LIN {X 0,Y 468.958,Z 580.155,A -85,B 0,C 180,E1 7791.266,E2 7791.266} C_VEL
LIN {X 0,Y 471.631,Z 601.526,A -85,B 0,C 180,E1 7791.982,E2 7791.982} C_VEL
LIN {X 0,Y 472.199,Z 602.706,A -85,B 0,C 180,E1 7792.061,E2 7792.061} C_VEL
LIN {X 0,Y 474.146,Z 606.908,A -85,B 0,C 180,E1 7792.333,E2 7792.333} C_VEL
LIN {X 0,Y 471.167,Z 650.181,A -85,B 0,C 180,E1 7793.72,E2 7793.72} C_VEL
LIN {X 0,Y 467.516,Z 690.525,A -85,B 0,C 180,E1 7795.792,E2 7795.792} C_VEL
LIN {X 0,Y 463.415,Z 728.527,A -85,B 0,C 180,E1 7798.596,E2 7798.596} C_VEL
LIN {X 0,Y 459.337,Z 761.729,A -85,B 0,C 180,E1 7801.949,E2 7801.949} C_VEL
LIN {X 0,Y 455.596,Z 791.466,A -85,B 0,C 180,E1 7805.971,E2 7805.971} C_VEL
LIN {X 0,Y 453.022,Z 813.983,A -85,B 0,C 180,E1 7810.044,E2 7810.044} C_VEL
LIN {X 0,Y 451.113,Z 833.292,A -85,B 0,C 180,E1 7814.929,E2 7814.929} C_VEL
LIN {X 0,Y 450.241,Z 846.703,A -85,B 0,C 180,E1 7819.864,E2 7819.864} C_VEL
LIN {X 0,Y 449.873,Z 853.995,A -85,B 0,C 180,E1 7824.224,E2 7824.224} C_VEL
LIN {X 0,Y 449.824,Z 857.107,A -85,B 0,C 180,E1 7828.077,E2 7828.077} C_VEL
LIN {X 0,Y 449.891,Z 857.107,A -85,B 0,C 180,E1 7831.922,E2 7831.922} C_VEL
LIN {X 0,Y 449.937,Z 852.735,A -85,B 0,C 180,E1 7836.742,E2 7836.742} C_VEL
LIN {X 0,Y 450.323,Z 843.318,A -85,B 0,C 180,E1 7841.6,E2 7841.6} C_VEL
LIN {X 0,Y 451.564,Z 828.297,A -85,B 0,C 180,E1 7846.503,E2 7846.503} C_VEL
LIN {X 0,Y 453.78,Z 807.486,A -85,B 0,C 180,E1 7851.27,E2 7851.27} C_VEL
LIN {X 0,Y 456.823,Z 782.083,A -85,B 0,C 180,E1 7855.434,E2 7855.434} C_VEL
LIN {X 0,Y 460.733,Z 750.709,A -85,B 0,C 180,E1 7859.294,E2 7859.294} C_VEL
LIN {X 0,Y 464.827,Z 716.248,A -85,B 0,C 180,E1 7862.435,E2 7862.435} C_VEL
LIN {X 0,Y 468.904,Z 677.165,A -85,B 0,C 180,E1 7865.008,E2 7865.008} C_VEL
LIN {X 0,Y 472.359,Z 635.769,A -85,B 0,C 180,E1 7866.854,E2 7866.854} C_VEL
LIN {X 0,Y 474.176,Z 604.683,A -85,B 0,C 180,E1 7867.761,E2 7867.761} C_VEL
LIN {X 0,Y 463.084,Z 582.313,A -85,B 0,C 180,E1 7869.225,E2 7869.225} C_VEL
LIN {X 0,Y 450.506,Z 554.48,A -85,B 0,C 180,E1 7870.935,E2 7870.935} C_VEL
LIN {X 0,Y 448.762,Z 549.53,A -85,B 0,C 180,E1 7871.266,E2 7871.266} C_VEL
LIN {X 0,Y 448.738,Z 549.53,A -85,B 0,C 180,E1 7877.741,E2 7877.741} C_VEL
LIN {X 0,Y 448.735,Z 549.53,A -85,B 0,C 180,E1 7883.819,E2 7883.819} C_VEL
LIN {X 0,Y 448.758,Z 549.53,A -85,B 0,C 180,E1 7889.713,E2 7889.713} C_VEL
LIN {X 0,Y 449.087,Z 549.53,A -85,B 0,C 180,E1 7895.084,E2 7895.084} C_VEL
LIN {X 0,Y 455.62,Z 577.259,A -85,B 0,C 180,E1 7895.913,E2 7895.913} C_VEL
LIN {X 0,Y 455.731,Z 612.964,A -85,B 0,C 180,E1 7896.707,E2 7896.707} C_VEL
LIN {X 0,Y 455.247,Z 640.891,A -85,B 0,C 180,E1 7898.053,E2 7898.053} C_VEL
LIN {X 0,Y 454.424,Z 665.309,A -85,B 0,C 180,E1 7899.978,E2 7899.978} C_VEL
LIN {X 0,Y 453.379,Z 686.918,A -85,B 0,C 180,E1 7902.574,E2 7902.574} C_VEL
LIN {X 0,Y 452.429,Z 703.348,A -85,B 0,C 180,E1 7905.55,E2 7905.55} C_VEL
LIN {X 0,Y 451.8,Z 714.901,A -85,B 0,C 180,E1 7908.932,E2 7908.932} C_VEL
LIN {X 0,Y 451.334,Z 720.778,A -85,B 0,C 180,E1 7912.319,E2 7912.319} C_VEL
LIN {X 0,Y 451.289,Z 721.854,A -85,B 0,C 180,E1 7914.247,E2 7914.247} C_VEL
LIN {X 0,Y 451.353,Z 719.256,A -85,B 0,C 180,E1 7918.088,E2 7918.088} C_VEL
LIN {X 0,Y 451.552,Z 711.787,A -85,B 0,C 180,E1 7921.441,E2 7921.441} C_VEL
LIN {X 0,Y 452.123,Z 698.574,A -85,B 0,C 180,E1 7924.791,E2 7924.791} C_VEL
LIN {X 0,Y 453.034,Z 679.581,A -85,B 0,C 180,E1 7927.902,E2 7927.902} C_VEL
LIN {X 0,Y 454.147,Z 656.595,A -85,B 0,C 180,E1 7930.414,E2 7930.414} C_VEL
LIN {X 0,Y 455.092,Z 630.622,A -85,B 0,C 180,E1 7932.301,E2 7932.301} C_VEL
LIN {X 0,Y 455.759,Z 601.099,A -85,B 0,C 180,E1 7933.569,E2 7933.569} C_VEL
LIN {X 0,Y 455.219,Z 572.995,A -85,B 0,C 180,E1 7934.176,E2 7934.176} C_VEL
LIN {X 0,Y 449.385,Z 549.53,A -85,B 0,C 180,E1 7934.829,E2 7934.829} C_VEL
LIN {X 0,Y 449.088,Z 549.53,A -85,B 0,C 180,E1 7941.697,E2 7941.697} C_VEL
LIN {X 0,Y 448.832,Z 549.53,A -85,B 0,C 180,E1 7948.085,E2 7948.085} C_VEL
LIN {X 0,Y 448.654,Z 549.53,A -85,B 0,C 180,E1 7954.88,E2 7954.88} C_VEL
LIN {X 0,Y 448.63,Z 549.53,A -85,B 0,C 180,E1 7959.73,E2 7959.73} C_VEL
LIN {X 0,Y 448.64,Z 549.53,A -85,B 0,C 180,E1 7965.056,E2 7965.056} C_VEL
LIN {X 0,Y 448.75,Z 549.53,A -85,B 0,C 180,E1 7970.67,E2 7970.67} C_VEL
LIN {X 0,Y 448.66,Z 549.53,A -85,B 0,C 180,E1 7977.439,E2 7977.439} C_VEL
LIN {X 0,Y 448.809,Z 550.244,A -85,B 0,C 180,E1 7978.288,E2 7978.288} C_VEL
LIN {X 0,Y 466.178,Z 592.56,A -85,B 0,C 180,E1 7981.008,E2 7981.008} C_VEL
LIN {X 0,Y 467.014,Z 599.43,A -85,B 0,C 180,E1 7981.357,E2 7981.357} C_VEL
LIN {X 0,Y 464.255,Z 634.875,A -85,B 0,C 180,E1 7983.149,E2 7983.149} C_VEL
LIN {X 0,Y 460.847,Z 669.201,A -85,B 0,C 180,E1 7985.708,E2 7985.708} C_VEL
LIN {X 0,Y 457.423,Z 699.289,A -85,B 0,C 180,E1 7988.847,E2 7988.847} C_VEL
LIN {X 0,Y 454.361,Z 725.705,A -85,B 0,C 180,E1 7992.607,E2 7992.607} C_VEL
LIN {X 0,Y 452.034,Z 746.654,A -85,B 0,C 180,E1 7996.731,E2 7996.731} C_VEL
LIN {X 0,Y 450.782,Z 761.886,A -85,B 0,C 180,E1 8000.97,E2 8000.97} C_VEL
LIN {X 0,Y 450.248,Z 771.956,A -85,B 0,C 180,E1 8005.193,E2 8005.193} C_VEL
LIN {X 0,Y 450.095,Z 778.035,A -85,B 0,C 180,E1 8010,E2 8010} C_VEL
LIN {X 0,Y 449.947,Z 778.916,A -85,B 0,C 180,E1 8013.847,E2 8013.847} C_VEL
LIN {X 0,Y 450.055,Z 775.148,A -85,B 0,C 180,E1 8018.76,E2 8018.76} C_VEL
LIN {X 0,Y 450.524,Z 765.71,A -85,B 0,C 180,E1 8023.562,E2 8023.562} C_VEL
LIN {X 0,Y 451.729,Z 751.367,A -85,B 0,C 180,E1 8028.026,E2 8028.026} C_VEL
LIN {X 0,Y 453.702,Z 731.868,A -85,B 0,C 180,E1 8032.233,E2 8032.233} C_VEL
LIN {X 0,Y 456.508,Z 707.237,A -85,B 0,C 180,E1 8036.053,E2 8036.053} C_VEL
LIN {X 0,Y 459.807,Z 678.331,A -85,B 0,C 180,E1 8039.359,E2 8039.359} C_VEL
LIN {X 0,Y 463.326,Z 644.876,A -85,B 0,C 180,E1 8042.126,E2 8042.126} C_VEL
LIN {X 0,Y 466.437,Z 608.507,A -85,B 0,C 180,E1 8044.2,E2 8044.2} C_VEL
LIN {X 0,Y 466.662,Z 594.193,A -85,B 0,C 180,E1 8044.838,E2 8044.838} C_VEL
LIN {X 0,Y 453.477,Z 560.1,A -85,B 0,C 180,E1 8047.08,E2 8047.08} C_VEL
LIN {X 0,Y 448.888,Z 549.53,A -85,B 0,C 180,E1 8047.902,E2 8047.902} C_VEL
LIN {X 0,Y 448.628,Z 549.53,A -85,B 0,C 180,E1 8055.054,E2 8055.054} C_VEL
LIN {X 0,Y 448.8,Z 549.53,A -85,B 0,C 180,E1 8060.663,E2 8060.663} C_VEL
LIN {X 0,Y 448.849,Z 549.53,A -85,B 0,C 180,E1 8067.202,E2 8067.202} C_VEL
LIN {X 0,Y 448.843,Z 549.53,A -85,B 0,C 180,E1 8074.078,E2 8074.078} C_VEL
LIN {X 0,Y 449.012,Z 549.53,A -85,B 0,C 180,E1 8078.739,E2 8078.739} C_VEL
LIN {X 0,Y 454.538,Z 576.815,A -85,B 0,C 180,E1 8079.412,E2 8079.412} C_VEL
LIN {X 0,Y 454.441,Z 624.708,A -85,B 0,C 180,E1 8080.368,E2 8080.368} C_VEL
LIN {X 0,Y 453.943,Z 650.535,A -85,B 0,C 180,E1 8081.607,E2 8081.607} C_VEL
LIN {X 0,Y 453.192,Z 674.327,A -85,B 0,C 180,E1 8083.554,E2 8083.554} C_VEL
LIN {X 0,Y 452.281,Z 694.707,A -85,B 0,C 180,E1 8086.171,E2 8086.171} C_VEL
LIN {X 0,Y 451.81,Z 708.538,A -85,B 0,C 180,E1 8088.923,E2 8088.923} C_VEL
LIN {X 0,Y 451.452,Z 717.552,A -85,B 0,C 180,E1 8091.839,E2 8091.839} C_VEL
LIN {X 0,Y 451.351,Z 721.412,A -85,B 0,C 180,E1 8094.239,E2 8094.239} C_VEL
LIN {X 0,Y 451.349,Z 722.421,A -85,B 0,C 180,E1 8096.162,E2 8096.162} C_VEL
LIN {X 0,Y 451.475,Z 720.452,A -85,B 0,C 180,E1 8099.038,E2 8099.038} C_VEL
LIN {X 0,Y 451.94,Z 712.572,A -85,B 0,C 180,E1 8102.388,E2 8102.388} C_VEL
LIN {X 0,Y 452.653,Z 700.047,A -85,B 0,C 180,E1 8105.256,E2 8105.256} C_VEL
LIN {X 0,Y 453.465,Z 681.764,A -85,B 0,C 180,E1 8107.886,E2 8107.886} C_VEL
LIN {X 0,Y 454.249,Z 659.647,A -85,B 0,C 180,E1 8109.914,E2 8109.914} C_VEL
LIN {X 0,Y 454.624,Z 634.95,A -85,B 0,C 180,E1 8111.285,E2 8111.285} C_VEL
LIN {X 0,Y 454.621,Z 605.314,A -85,B 0,C 180,E1 8112.05,E2 8112.05} C_VEL
LIN {X 0,Y 454.181,Z 569.256,A -85,B 0,C 180,E1 8112.708,E2 8112.708} C_VEL
LIN {X 0,Y 449.327,Z 549.53,A -85,B 0,C 180,E1 8113.328,E2 8113.328} C_VEL
LIN {X 0,Y 449.048,Z 549.53,A -85,B 0,C 180,E1 8119.773,E2 8119.773} C_VEL
LIN {X 0,Y 448.861,Z 549.53,A -85,B 0,C 180,E1 8125.911,E2 8125.911} C_VEL
LIN {X 0,Y 448.646,Z 549.53,A -85,B 0,C 180,E1 8132.757,E2 8132.757} C_VEL
LIN {X 0,Y 448.756,Z 549.53,A -85,B 0,C 180,E1 8139.331,E2 8139.331} C_VEL
LIN {X 0,Y 448.66,Z 549.53,A -85,B 0,C 180,E1 8145.058,E2 8145.058} C_VEL
LIN {X 0,Y 448.725,Z 549.68,A -85,B 0,C 180,E1 8148.7,E2 8148.7} C_VEL
LIN {X 0,Y 453.525,Z 559.924,A -85,B 0,C 180,E1 8149.401,E2 8149.401} C_VEL
LIN {X 0,Y 470.3,Z 599.601,A -85,B 0,C 180,E1 8151.819,E2 8151.819} C_VEL
LIN {X 0,Y 472.199,Z 602.706,A -85,B 0,C 180,E1 8152.061,E2 8152.061} C_VEL
LIN {X 0,Y 472.315,Z 609.467,A -85,B 0,C 180,E1 8152.253,E2 8152.253} C_VEL
LIN {X 0,Y 466.587,Z 624.047,A -85,B 0,C 180,E1 8152.272,E2 8152.272} C_VEL
LIN {X 0,Y 466.404,Z 625.593,A -85,B 0,C 180,E1 8152.315,E2 8152.315} C_VEL
LIN {X 0,Y 462.996,Z 666.329,A -85,B 0,C 180,E1 8153.961,E2 8153.961} C_VEL
LIN {X 0,Y 458.94,Z 704.99,A -85,B 0,C 180,E1 8156.282,E2 8156.282} C_VEL
LIN {X 0,Y 454.394,Z 742.555,A -85,B 0,C 180,E1 8159.469,E2 8159.469} C_VEL
LIN {X 0,Y 450.434,Z 773.095,A -85,B 0,C 180,E1 8162.997,E2 8162.997} C_VEL
LIN {X 0,Y 446.719,Z 801.611,A -85,B 0,C 180,E1 8167.4,E2 8167.4} C_VEL
LIN {X 0,Y 444.117,Z 824.449,A -85,B 0,C 180,E1 8172.191,E2 8172.191} C_VEL
LIN {X 0,Y 442.649,Z 840.782,A -85,B 0,C 180,E1 8177.196,E2 8177.196} C_VEL
LIN {X 0,Y 442.08,Z 851.261,A -85,B 0,C 180,E1 8182.151,E2 8182.151} C_VEL
LIN {X 0,Y 441.884,Z 855.94,A -85,B 0,C 180,E1 8186.083,E2 8186.083} C_VEL
LIN {X 0,Y 441.939,Z 857.5,A -85,B 0,C 180,E1 8190,E2 8190} C_VEL
LIN {X 0,Y 441.903,Z 855.94,A -85,B 0,C 180,E1 8193.916,E2 8193.916} C_VEL
LIN {X 0,Y 442.182,Z 849.486,A -85,B 0,C 180,E1 8198.894,E2 8198.894} C_VEL
LIN {X 0,Y 442.989,Z 836.944,A -85,B 0,C 180,E1 8204.165,E2 8204.165} C_VEL
LIN {X 0,Y 444.463,Z 821.337,A -85,B 0,C 180,E1 8208.564,E2 8208.564} C_VEL
LIN {X 0,Y 447.229,Z 797.324,A -85,B 0,C 180,E1 8213.359,E2 8213.359} C_VEL
LIN {X 0,Y 451.125,Z 768.092,A -85,B 0,C 180,E1 8217.665,E2 8217.665} C_VEL
LIN {X 0,Y 455.3,Z 736.094,A -85,B 0,C 180,E1 8221.167,E2 8221.167} C_VEL
LIN {X 0,Y 459.557,Z 700.748,A -85,B 0,C 180,E1 8224.023,E2 8224.023} C_VEL
LIN {X 0,Y 463.565,Z 661.836,A -85,B 0,C 180,E1 8226.279,E2 8226.279} C_VEL
LIN {X 0,Y 466.918,Z 621.282,A -85,B 0,C 180,E1 8227.832,E2 8227.832} C_VEL
LIN {X 0,Y 467.172,Z 607.41,A -85,B 0,C 180,E1 8228.257,E2 8228.257} C_VEL
LIN {X 0,Y 455.657,Z 582.229,A -85,B 0,C 180,E1 8229.897,E2 8229.897} C_VEL
LIN {X 0,Y 442.976,Z 554.912,A -85,B 0,C 180,E1 8231.669,E2 8231.669} C_VEL
LIN {X 0,Y 440.83,Z 549.53,A -85,B 0,C 180,E1 8232.063,E2 8232.063} C_VEL
LIN {X 0,Y 440.77,Z 549.53,A -85,B 0,C 180,E1 8238.874,E2 8238.874} C_VEL
LIN {X 0,Y 440.809,Z 549.53,A -85,B 0,C 180,E1 8245.253,E2 8245.253} C_VEL
LIN {X 0,Y 440.892,Z 549.53,A -85,B 0,C 180,E1 8251.374,E2 8251.374} C_VEL
LIN {X 0,Y 441.126,Z 549.809,A -85,B 0,C 180,E1 8254.732,E2 8254.732} C_VEL
LIN {X 0,Y 448.163,Z 578.479,A -85,B 0,C 180,E1 8255.616,E2 8255.616} C_VEL
LIN {X 0,Y 448.252,Z 614.662,A -85,B 0,C 180,E1 8256.441,E2 8256.441} C_VEL
LIN {X 0,Y 447.746,Z 642.172,A -85,B 0,C 180,E1 8257.782,E2 8257.782} C_VEL
LIN {X 0,Y 446.889,Z 666.849,A -85,B 0,C 180,E1 8259.755,E2 8259.755} C_VEL
LIN {X 0,Y 445.835,Z 687.649,A -85,B 0,C 180,E1 8262.269,E2 8262.269} C_VEL
LIN {X 0,Y 444.822,Z 704.385,A -85,B 0,C 180,E1 8265.297,E2 8265.297} C_VEL
LIN {X 0,Y 444.113,Z 716.107,A -85,B 0,C 180,E1 8268.738,E2 8268.738} C_VEL
LIN {X 0,Y 443.58,Z 722.102,A -85,B 0,C 180,E1 8272.184,E2 8272.184} C_VEL
LIN {X 0,Y 443.521,Z 723.232,A -85,B 0,C 180,E1 8274.146,E2 8274.146} C_VEL
LIN {X 0,Y 443.592,Z 720.65,A -85,B 0,C 180,E1 8278.055,E2 8278.055} C_VEL
LIN {X 0,Y 443.789,Z 713.177,A -85,B 0,C 180,E1 8281.466,E2 8281.466} C_VEL
LIN {X 0,Y 444.372,Z 699.941,A -85,B 0,C 180,E1 8284.875,E2 8284.875} C_VEL
LIN {X 0,Y 445.316,Z 680.911,A -85,B 0,C 180,E1 8288.04,E2 8288.04} C_VEL
LIN {X 0,Y 446.47,Z 657.872,A -85,B 0,C 180,E1 8290.595,E2 8290.595} C_VEL
LIN {X 0,Y 447.489,Z 630.925,A -85,B 0,C 180,E1 8292.567,E2 8292.567} C_VEL
LIN {X 0,Y 448.18,Z 601.127,A -85,B 0,C 180,E1 8293.844,E2 8293.844} C_VEL
LIN {X 0,Y 447.583,Z 573.933,A -85,B 0,C 180,E1 8294.438,E2 8294.438} C_VEL
LIN {X 0,Y 441.441,Z 549.53,A -85,B 0,C 180,E1 8295.121,E2 8295.121} C_VEL
LIN {X 0,Y 441.119,Z 549.53,A -85,B 0,C 180,E1 8302.11,E2 8302.11} C_VEL
LIN {X 0,Y 440.911,Z 549.53,A -85,B 0,C 180,E1 8308.635,E2 8308.635} C_VEL
LIN {X 0,Y 440.731,Z 549.53,A -85,B 0,C 180,E1 8315.602,E2 8315.602} C_VEL
LIN {X 0,Y 440.614,Z 549.53,A -85,B 0,C 180,E1 8321.103,E2 8321.103} C_VEL
LIN {X 0,Y 440.674,Z 549.53,A -85,B 0,C 180,E1 8326.769,E2 8326.769} C_VEL
LIN {X 0,Y 440.771,Z 549.53,A -85,B 0,C 180,E1 8331.953,E2 8331.953} C_VEL
LIN {X 0,Y 440.806,Z 550.142,A -85,B 0,C 180,E1 8337.555,E2 8337.555} C_VEL
LIN {X 0,Y 457.96,Z 591.22,A -85,B 0,C 180,E1 8340.312,E2 8340.312} C_VEL
LIN {X 0,Y 460.191,Z 600.559,A -85,B 0,C 180,E1 8340.887,E2 8340.887} C_VEL
LIN {X 0,Y 457.232,Z 636.395,A -85,B 0,C 180,E1 8342.744,E2 8342.744} C_VEL
LIN {X 0,Y 453.677,Z 669.986,A -85,B 0,C 180,E1 8345.298,E2 8345.298} C_VEL
LIN {X 0,Y 450.19,Z 698.924,A -85,B 0,C 180,E1 8348.362,E2 8348.362} C_VEL
LIN {X 0,Y 446.944,Z 725.067,A -85,B 0,C 180,E1 8352.087,E2 8352.087} C_VEL
LIN {X 0,Y 444.456,Z 746.31,A -85,B 0,C 180,E1 8356.25,E2 8356.25} C_VEL
LIN {X 0,Y 442.984,Z 762.695,A -85,B 0,C 180,E1 8360.832,E2 8360.832} C_VEL
LIN {X 0,Y 442.398,Z 772.708,A -85,B 0,C 180,E1 8365.108,E2 8365.108} C_VEL
LIN {X 0,Y 442.246,Z 778.766,A -85,B 0,C 180,E1 8370,E2 8370} C_VEL
LIN {X 0,Y 442.09,Z 779.613,A -85,B 0,C 180,E1 8373.915,E2 8373.915} C_VEL
LIN {X 0,Y 442.22,Z 775.839,A -85,B 0,C 180,E1 8378.855,E2 8378.855} C_VEL
LIN {X 0,Y 442.67,Z 767.491,A -85,B 0,C 180,E1 8383.301,E2 8383.301} C_VEL
LIN {X 0,Y 443.856,Z 753.673,A -85,B 0,C 180,E1 8387.82,E2 8387.82} C_VEL
LIN {X 0,Y 445.91,Z 734.596,A -85,B 0,C 180,E1 8392.119,E2 8392.119} C_VEL
LIN {X 0,Y 448.796,Z 710.116,A -85,B 0,C 180,E1 8396.102,E2 8396.102} C_VEL
LIN {X 0,Y 452.409,Z 680.764,A -85,B 0,C 180,E1 8399.601,E2 8399.601} C_VEL
LIN {X 0,Y 456.178,Z 647.674,A -85,B 0,C 180,E1 8402.448,E2 8402.448} C_VEL
LIN {X 0,Y 459.521,Z 612.087,A -85,B 0,C 180,E1 8404.563,E2 8404.563} C_VEL
LIN {X 0,Y 459.83,Z 596.401,A -85,B 0,C 180,E1 8405.302,E2 8405.302} C_VEL
LIN {X 0,Y 447.484,Z 564.002,A -85,B 0,C 180,E1 8407.525,E2 8407.525} C_VEL
LIN {X 0,Y 440.941,Z 549.53,A -85,B 0,C 180,E1 8408.628,E2 8408.628} C_VEL
LIN {X 0,Y 440.65,Z 549.53,A -85,B 0,C 180,E1 8415.991,E2 8415.991} C_VEL
LIN {X 0,Y 440.881,Z 549.53,A -85,B 0,C 180,E1 8421.963,E2 8421.963} C_VEL
LIN {X 0,Y 440.923,Z 549.53,A -85,B 0,C 180,E1 8426.793,E2 8426.793} C_VEL
LIN {X 0,Y 440.882,Z 549.53,A -85,B 0,C 180,E1 8433.574,E2 8433.574} C_VEL
LIN {X 0,Y 441.08,Z 549.53,A -85,B 0,C 180,E1 8438.424,E2 8438.424} C_VEL
LIN {X 0,Y 446.961,Z 578.421,A -85,B 0,C 180,E1 8439.19,E2 8439.19} C_VEL
LIN {X 0,Y 446.777,Z 625.969,A -85,B 0,C 180,E1 8440.16,E2 8440.16} C_VEL
LIN {X 0,Y 446.244,Z 652.884,A -85,B 0,C 180,E1 8441.495,E2 8441.495} C_VEL
LIN {X 0,Y 445.445,Z 676.631,A -85,B 0,C 180,E1 8443.513,E2 8443.513} C_VEL
LIN {X 0,Y 444.553,Z 695.54,A -85,B 0,C 180,E1 8445.986,E2 8445.986} C_VEL
LIN {X 0,Y 444.065,Z 709.321,A -85,B 0,C 180,E1 8448.728,E2 8448.728} C_VEL
LIN {X 0,Y 443.704,Z 717.704,A -85,B 0,C 180,E1 8451.325,E2 8451.325} C_VEL
LIN {X 0,Y 443.582,Z 722.615,A -85,B 0,C 180,E1 8454.138,E2 8454.138} C_VEL
LIN {X 0,Y 443.582,Z 723.739,A -85,B 0,C 180,E1 8456.094,E2 8456.094} C_VEL
LIN {X 0,Y 443.706,Z 721.914,A -85,B 0,C 180,E1 8459.021,E2 8459.021} C_VEL
LIN {X 0,Y 444.218,Z 714.183,A -85,B 0,C 180,E1 8462.429,E2 8462.429} C_VEL
LIN {X 0,Y 444.974,Z 701.791,A -85,B 0,C 180,E1 8465.347,E2 8465.347} C_VEL
LIN {X 0,Y 445.847,Z 683.655,A -85,B 0,C 180,E1 8468.021,E2 8468.021} C_VEL
LIN {X 0,Y 446.623,Z 661.695,A -85,B 0,C 180,E1 8470.09,E2 8470.09} C_VEL
LIN {X 0,Y 447.066,Z 635.885,A -85,B 0,C 180,E1 8471.549,E2 8471.549} C_VEL
LIN {X 0,Y 447.075,Z 605.219,A -85,B 0,C 180,E1 8472.339,E2 8472.339} C_VEL
LIN {X 0,Y 446.826,Z 571.258,A -85,B 0,C 180,E1 8472.971,E2 8472.971} C_VEL
LIN {X 0,Y 441.397,Z 549.53,A -85,B 0,C 180,E1 8473.636,E2 8473.636} C_VEL
LIN {X 0,Y 441.132,Z 549.53,A -85,B 0,C 180,E1 8479.999,E2 8479.999} C_VEL
LIN {X 0,Y 440.879,Z 549.53,A -85,B 0,C 180,E1 8486.416,E2 8486.416} C_VEL
LIN {X 0,Y 440.704,Z 549.53,A -85,B 0,C 180,E1 8493.215,E2 8493.215} C_VEL
LIN {X 0,Y 440.787,Z 549.53,A -85,B 0,C 180,E1 8498.049,E2 8498.049} C_VEL
LIN {X 0,Y 440.686,Z 549.53,A -85,B 0,C 180,E1 8504.014,E2 8504.014} C_VEL
LIN {X 0,Y 440.783,Z 549.53,A -85,B 0,C 180,E1 8507.826,E2 8507.826} C_VEL
LIN {X 0,Y 445.066,Z 559.069,A -85,B 0,C 180,E1 8508.506,E2 8508.506} C_VEL
LIN {X 0,Y 453.835,Z 578.128,A -85,B 0,C 180,E1 8509.804,E2 8509.804} C_VEL
LIN {X 0,Y 464.775,Z 604.46,A -85,B 0,C 180,E1 8511.477,E2 8511.477} C_VEL
LIN {X 0,Y 467.444,Z 608.833,A -85,B 0,C 180,E1 8511.828,E2 8511.828} C_VEL
LIN {X 0,Y 466.404,Z 625.593,A -85,B 0,C 180,E1 8512.315,E2 8512.315} C_VEL
LIN {X 0,Y 461.732,Z 642.303,A -85,B 0,C 180,E1 8512.633,E2 8512.633} C_VEL
LIN {X 0,Y 457.12,Z 656.694,A -85,B 0,C 180,E1 8512.98,E2 8512.98} C_VEL
LIN {X 0,Y 456.86,Z 658.754,A -85,B 0,C 180,E1 8513.069,E2 8513.069} C_VEL
LIN {X 0,Y 452.474,Z 700.061,A -85,B 0,C 180,E1 8515.457,E2 8515.457} C_VEL
LIN {X 0,Y 447.896,Z 737.285,A -85,B 0,C 180,E1 8518.515,E2 8518.515} C_VEL
LIN {X 0,Y 443.641,Z 768.24,A -85,B 0,C 180,E1 8521.981,E2 8521.981} C_VEL
LIN {X 0,Y 439.677,Z 796.512,A -85,B 0,C 180,E1 8526.214,E2 8526.214} C_VEL
LIN {X 0,Y 436.742,Z 820.602,A -85,B 0,C 180,E1 8531.097,E2 8531.097} C_VEL
LIN {X 0,Y 434.988,Z 838.73,A -85,B 0,C 180,E1 8536.234,E2 8536.234} C_VEL
LIN {X 0,Y 434.288,Z 849.592,A -85,B 0,C 180,E1 8541.003,E2 8541.003} C_VEL
LIN {X 0,Y 434.002,Z 855.939,A -85,B 0,C 180,E1 8546.012,E2 8546.012} C_VEL
LIN {X 0,Y 434.039,Z 857.5,A -85,B 0,C 180,E1 8550,E2 8550} C_VEL
LIN {X 0,Y 434.021,Z 855.939,A -85,B 0,C 180,E1 8553.987,E2 8553.987} C_VEL
LIN {X 0,Y 434.288,Z 849.594,A -85,B 0,C 180,E1 8558.996,E2 8558.996} C_VEL
LIN {X 0,Y 435.088,Z 837.877,A -85,B 0,C 180,E1 8564.052,E2 8564.052} C_VEL
LIN {X 0,Y 436.836,Z 819.531,A -85,B 0,C 180,E1 8569.16,E2 8569.16} C_VEL
LIN {X 0,Y 439.656,Z 796.582,A -85,B 0,C 180,E1 8573.786,E2 8573.786} C_VEL
LIN {X 0,Y 443.666,Z 768.377,A -85,B 0,C 180,E1 8578.016,E2 8578.016} C_VEL
LIN {X 0,Y 447.921,Z 737.455,A -85,B 0,C 180,E1 8581.482,E2 8581.482} C_VEL
LIN {X 0,Y 452.467,Z 702.018,A -85,B 0,C 180,E1 8584.426,E2 8584.426} C_VEL
LIN {X 0,Y 456.624,Z 663.574,A -85,B 0,C 180,E1 8586.713,E2 8586.713} C_VEL
LIN {X 0,Y 460.316,Z 621.55,A -85,B 0,C 180,E1 8588.364,E2 8588.364} C_VEL
LIN {X 0,Y 460.446,Z 610.446,A -85,B 0,C 180,E1 8588.732,E2 8588.732} C_VEL
LIN {X 0,Y 448.851,Z 583.513,A -85,B 0,C 180,E1 8590.505,E2 8590.505} C_VEL
LIN {X 0,Y 436.391,Z 557.835,A -85,B 0,C 180,E1 8592.283,E2 8592.283} C_VEL
LIN {X 0,Y 432.841,Z 549.53,A -85,B 0,C 180,E1 8592.941,E2 8592.941} C_VEL
LIN {X 0,Y 432.825,Z 549.53,A -85,B 0,C 180,E1 8598.521,E2 8598.521} C_VEL
LIN {X 0,Y 432.835,Z 549.53,A -85,B 0,C 180,E1 8603.658,E2 8603.658} C_VEL
LIN {X 0,Y 432.881,Z 549.53,A -85,B 0,C 180,E1 8610.643,E2 8610.643} C_VEL
LIN {X 0,Y 433.162,Z 549.53,A -85,B 0,C 180,E1 8614.303,E2 8614.303} C_VEL
LIN {X 0,Y 440.728,Z 579.778,A -85,B 0,C 180,E1 8615.301,E2 8615.301} C_VEL
LIN {X 0,Y 440.78,Z 616.347,A -85,B 0,C 180,E1 8616.154,E2 8616.154} C_VEL
LIN {X 0,Y 440.254,Z 645.272,A -85,B 0,C 180,E1 8617.616,E2 8617.616} C_VEL
LIN {X 0,Y 439.278,Z 670.948,A -85,B 0,C 180,E1 8619.782,E2 8619.782} C_VEL
LIN {X 0,Y 438.108,Z 691.789,A -85,B 0,C 180,E1 8622.464,E2 8622.464} C_VEL
LIN {X 0,Y 437.01,Z 708.322,A -85,B 0,C 180,E1 8625.729,E2 8625.729} C_VEL
LIN {X 0,Y 436.35,Z 718.588,A -85,B 0,C 180,E1 8629.04,E2 8629.04} C_VEL
LIN {X 0,Y 435.828,Z 723.442,A -85,B 0,C 180,E1 8632.044,E2 8632.044} C_VEL
LIN {X 0,Y 435.743,Z 724.604,A -85,B 0,C 180,E1 8634.041,E2 8634.041} C_VEL
LIN {X 0,Y 435.779,Z 723.27,A -85,B 0,C 180,E1 8637.027,E2 8637.027} C_VEL
LIN {X 0,Y 435.907,Z 717.221,A -85,B 0,C 180,E1 8640.5,E2 8640.5} C_VEL
LIN {X 0,Y 436.422,Z 705.775,A -85,B 0,C 180,E1 8643.97,E2 8643.97} C_VEL
LIN {X 0,Y 437.261,Z 688.914,A -85,B 0,C 180,E1 8647.191,E2 8647.191} C_VEL
LIN {X 0,Y 438.388,Z 667.876,A -85,B 0,C 180,E1 8649.915,E2 8649.915} C_VEL
LIN {X 0,Y 439.504,Z 642.176,A -85,B 0,C 180,E1 8652.145,E2 8652.145} C_VEL
LIN {X 0,Y 440.406,Z 613.587,A -85,B 0,C 180,E1 8653.693,E2 8653.693} C_VEL
LIN {X 0,Y 440.767,Z 580.332,A -85,B 0,C 180,E1 8654.57,E2 8654.57} C_VEL
LIN {X 0,Y 433.502,Z 549.53,A -85,B 0,C 180,E1 8655.471,E2 8655.471} C_VEL
LIN {X 0,Y 433.183,Z 549.53,A -85,B 0,C 180,E1 8662.537,E2 8662.537} C_VEL
LIN {X 0,Y 432.894,Z 549.53,A -85,B 0,C 180,E1 8669.36,E2 8669.36} C_VEL
LIN {X 0,Y 432.823,Z 549.53,A -85,B 0,C 180,E1 8673.912,E2 8673.912} C_VEL
LIN {X 0,Y 432.657,Z 549.53,A -85,B 0,C 180,E1 8679.88,E2 8679.88} C_VEL
LIN {X 0,Y 432.741,Z 549.53,A -85,B 0,C 180,E1 8685.774,E2 8685.774} C_VEL
LIN {X 0,Y 432.763,Z 549.53,A -85,B 0,C 180,E1 8691.119,E2 8691.119} C_VEL
LIN {X 0,Y 432.875,Z 550.253,A -85,B 0,C 180,E1 8696.797,E2 8696.797} C_VEL
LIN {X 0,Y 450.238,Z 590.991,A -85,B 0,C 180,E1 8699.671,E2 8699.671} C_VEL
LIN {X 0,Y 453.385,Z 601.945,A -85,B 0,C 180,E1 8700.412,E2 8700.412} C_VEL
LIN {X 0,Y 450.283,Z 637.555,A -85,B 0,C 180,E1 8702.298,E2 8702.298} C_VEL
LIN {X 0,Y 446.554,Z 670.859,A -85,B 0,C 180,E1 8704.877,E2 8704.877} C_VEL
LIN {X 0,Y 442.59,Z 701.666,A -85,B 0,C 180,E1 8708.234,E2 8708.234} C_VEL
LIN {X 0,Y 439.254,Z 727.045,A -85,B 0,C 180,E1 8711.988,E2 8711.988} C_VEL
LIN {X 0,Y 436.674,Z 748.042,A -85,B 0,C 180,E1 8716.255,E2 8716.255} C_VEL
LIN {X 0,Y 435.142,Z 764.326,A -85,B 0,C 180,E1 8720.976,E2 8720.976} C_VEL
LIN {X 0,Y 434.562,Z 773.455,A -85,B 0,C 180,E1 8725.02,E2 8725.02} C_VEL
LIN {X 0,Y 434.382,Z 779.497,A -85,B 0,C 180,E1 8730,E2 8730} C_VEL
LIN {X 0,Y 434.213,Z 780.312,A -85,B 0,C 180,E1 8733.986,E2 8733.986} C_VEL
LIN {X 0,Y 434.36,Z 776.472,A -85,B 0,C 180,E1 8738.996,E2 8738.996} C_VEL
LIN {X 0,Y 434.91,Z 767.593,A -85,B 0,C 180,E1 8743.686,E2 8743.686} C_VEL
LIN {X 0,Y 436.165,Z 753.978,A -85,B 0,C 180,E1 8748.145,E2 8748.145} C_VEL
LIN {X 0,Y 438.349,Z 734.743,A -85,B 0,C 180,E1 8752.521,E2 8752.521} C_VEL
LIN {X 0,Y 441.656,Z 709.389,A -85,B 0,C 180,E1 8756.674,E2 8756.674} C_VEL
LIN {X 0,Y 445.474,Z 680.527,A -85,B 0,C 180,E1 8760.143,E2 8760.143} C_VEL
LIN {X 0,Y 449.419,Z 647.615,A -85,B 0,C 180,E1 8762.991,E2 8762.991} C_VEL
LIN {X 0,Y 452.837,Z 612.932,A -85,B 0,C 180,E1 8765.08,E2 8765.08} C_VEL
LIN {X 0,Y 453.234,Z 599.105,A -85,B 0,C 180,E1 8765.745,E2 8765.745} C_VEL
LIN {X 0,Y 441.659,Z 568.235,A -85,B 0,C 180,E1 8767.958,E2 8767.958} C_VEL
LIN {X 0,Y 432.941,Z 549.53,A -85,B 0,C 180,E1 8769.484,E2 8769.484} C_VEL
LIN {X 0,Y 432.728,Z 549.53,A -85,B 0,C 180,E1 8775.771,E2 8775.771} C_VEL
LIN {X 0,Y 432.869,Z 549.53,A -85,B 0,C 180,E1 8781.128,E2 8781.128} C_VEL
LIN {X 0,Y 433.045,Z 549.53,A -85,B 0,C 180,E1 8786.764,E2 8786.764} C_VEL
LIN {X 0,Y 432.976,Z 549.53,A -85,B 0,C 180,E1 8793.053,E2 8793.053} C_VEL
LIN {X 0,Y 433.145,Z 549.53,A -85,B 0,C 180,E1 8798.145,E2 8798.145} C_VEL
LIN {X 0,Y 439.232,Z 577.752,A -85,B 0,C 180,E1 8798.913,E2 8798.913} C_VEL
LIN {X 0,Y 439.136,Z 627.616,A -85,B 0,C 180,E1 8799.959,E2 8799.959} C_VEL
LIN {X 0,Y 438.556,Z 654.011,A -85,B 0,C 180,E1 8801.295,E2 8801.295} C_VEL
LIN {X 0,Y 437.737,Z 677.768,A -85,B 0,C 180,E1 8803.343,E2 8803.343} C_VEL
LIN {X 0,Y 436.783,Z 697.587,A -85,B 0,C 180,E1 8806,E2 8806} C_VEL
LIN {X 0,Y 436.24,Z 712.054,A -85,B 0,C 180,E1 8809.028,E2 8809.028} C_VEL
LIN {X 0,Y 435.8,Z 721.391,A -85,B 0,C 180,E1 8812.422,E2 8812.422} C_VEL
LIN {X 0,Y 435.811,Z 725.06,A -85,B 0,C 180,E1 8816.024,E2 8816.024} C_VEL
LIN {X 0,Y 435.959,Z 723.389,A -85,B 0,C 180,E1 8819.004,E2 8819.004} C_VEL
LIN {X 0,Y 436.504,Z 715.825,A -85,B 0,C 180,E1 8822.472,E2 8822.472} C_VEL
LIN {X 0,Y 437.281,Z 703.545,A -85,B 0,C 180,E1 8825.441,E2 8825.441} C_VEL
LIN {X 0,Y 438.22,Z 685.578,A -85,B 0,C 180,E1 8828.162,E2 8828.162} C_VEL
LIN {X 0,Y 439.061,Z 663.153,A -85,B 0,C 180,E1 8830.325,E2 8830.325} C_VEL
LIN {X 0,Y 439.537,Z 637.121,A -85,B 0,C 180,E1 8831.817,E2 8831.817} C_VEL
LIN {X 0,Y 439.523,Z 604.015,A -85,B 0,C 180,E1 8832.661,E2 8832.661} C_VEL
LIN {X 0,Y 439.068,Z 571.373,A -85,B 0,C 180,E1 8833.306,E2 8833.306} C_VEL
LIN {X 0,Y 433.411,Z 549.53,A -85,B 0,C 180,E1 8834.102,E2 8834.102} C_VEL
LIN {X 0,Y 433.18,Z 549.53,A -85,B 0,C 180,E1 8840.382,E2 8840.382} C_VEL
LIN {X 0,Y 432.955,Z 549.53,A -85,B 0,C 180,E1 8846.938,E2 8846.938} C_VEL
LIN {X 0,Y 432.807,Z 549.53,A -85,B 0,C 180,E1 8853.902,E2 8853.902} C_VEL
LIN {X 0,Y 432.766,Z 549.53,A -85,B 0,C 180,E1 8859.896,E2 8859.896} C_VEL
LIN {X 0,Y 432.778,Z 549.53,A -85,B 0,C 180,E1 8866.379,E2 8866.379} C_VEL
LIN {X 0,Y 432.791,Z 549.531,A -85,B 0,C 180,E1 8866.936,E2 8866.936} C_VEL
LIN {X 0,Y 435.183,Z 555.159,A -85,B 0,C 180,E1 8867.334,E2 8867.334} C_VEL
LIN {X 0,Y 446.252,Z 577.13,A -85,B 0,C 180,E1 8869.016,E2 8869.016} C_VEL
LIN {X 0,Y 458.627,Z 608.29,A -85,B 0,C 180,E1 8871.049,E2 8871.049} C_VEL
LIN {X 0,Y 460.755,Z 612.999,A -85,B 0,C 180,E1 8871.392,E2 8871.392} C_VEL
LIN {X 0,Y 456.984,Z 657.402,A -85,B 0,C 180,E1 8873.007,E2 8873.007} C_VEL
LIN {X 0,Y 456.86,Z 658.754,A -85,B 0,C 180,E1 8873.069,E2 8873.069} C_VEL
LIN {X 0,Y 451.965,Z 674.993,A -85,B 0,C 180,E1 8873.641,E2 8873.641} C_VEL
LIN {X 0,Y 446.703,Z 690.803,A -85,B 0,C 180,E1 8874.34,E2 8874.34} C_VEL
LIN {X 0,Y 442.073,Z 727.964,A -85,B 0,C 180,E1 8877.183,E2 8877.183} C_VEL
LIN {X 0,Y 437.392,Z 760.685,A -85,B 0,C 180,E1 8880.609,E2 8880.609} C_VEL
LIN {X 0,Y 433.142,Z 789.231,A -85,B 0,C 180,E1 8884.659,E2 8884.659} C_VEL
LIN {X 0,Y 429.68,Z 814.276,A -85,B 0,C 180,E1 8889.437,E2 8889.437} C_VEL
LIN {X 0,Y 427.527,Z 834.039,A -85,B 0,C 180,E1 8894.647,E2 8894.647} C_VEL
LIN {X 0,Y 426.596,Z 847.379,A -85,B 0,C 180,E1 8899.811,E2 8899.811} C_VEL
LIN {X 0,Y 426.191,Z 853.972,A -85,B 0,C 180,E1 8903.901,E2 8903.901} C_VEL
LIN {X 0,Y 426.108,Z 857.104,A -85,B 0,C 180,E1 8907.97,E2 8907.97} C_VEL
LIN {X 0,Y 426.17,Z 857.104,A -85,B 0,C 180,E1 8912.029,E2 8912.029} C_VEL
LIN {X 0,Y 426.3,Z 852.982,A -85,B 0,C 180,E1 8916.89,E2 8916.89} C_VEL
LIN {X 0,Y 426.808,Z 842.75,A -85,B 0,C 180,E1 8922.248,E2 8922.248} C_VEL
LIN {X 0,Y 428.216,Z 827.773,A -85,B 0,C 180,E1 8927.215,E2 8927.215} C_VEL
LIN {X 0,Y 430.742,Z 806.279,A -85,B 0,C 180,E1 8932.266,E2 8932.266} C_VEL
LIN {X 0,Y 434.569,Z 779.727,A -85,B 0,C 180,E1 8936.837,E2 8936.837} C_VEL
LIN {X 0,Y 438.951,Z 750.216,A -85,B 0,C 180,E1 8940.628,E2 8940.628} C_VEL
LIN {X 0,Y 443.665,Z 716.165,A -85,B 0,C 180,E1 8943.85,E2 8943.85} C_VEL
LIN {X 0,Y 448.286,Z 677.495,A -85,B 0,C 180,E1 8946.488,E2 8946.488} C_VEL
LIN {X 0,Y 452.538,Z 634.161,A -85,B 0,C 180,E1 8948.495,E2 8948.495} C_VEL
LIN {X 0,Y 453.716,Z 613.311,A -85,B 0,C 180,E1 8949.206,E2 8949.206} C_VEL
LIN {X 0,Y 440.3,Z 580.733,A -85,B 0,C 180,E1 8951.398,E2 8951.398} C_VEL
LIN {X 0,Y 424.952,Z 550.122,A -85,B 0,C 180,E1 8953.685,E2 8953.685} C_VEL
LIN {X 0,Y 424.896,Z 549.53,A -85,B 0,C 180,E1 8960.268,E2 8960.268} C_VEL
LIN {X 0,Y 424.866,Z 549.53,A -85,B 0,C 180,E1 8965.375,E2 8965.375} C_VEL
LIN {X 0,Y 425.058,Z 549.53,A -85,B 0,C 180,E1 8972.576,E2 8972.576} C_VEL
LIN {X 0,Y 425.22,Z 549.53,A -85,B 0,C 180,E1 8973.852,E2 8973.852} C_VEL
LIN {X 0,Y 433.206,Z 579.535,A -85,B 0,C 180,E1 8974.927,E2 8974.927} C_VEL
LIN {X 0,Y 433.343,Z 619.127,A -85,B 0,C 180,E1 8975.896,E2 8975.896} C_VEL
LIN {X 0,Y 432.793,Z 647.441,A -85,B 0,C 180,E1 8977.373,E2 8977.373} C_VEL
LIN {X 0,Y 431.753,Z 672.648,A -85,B 0,C 180,E1 8979.547,E2 8979.547} C_VEL
LIN {X 0,Y 430.59,Z 692.662,A -85,B 0,C 180,E1 8982.147,E2 8982.147} C_VEL
LIN {X 0,Y 429.413,Z 708.84,A -85,B 0,C 180,E1 8985.317,E2 8985.317} C_VEL
LIN {X 0,Y 428.64,Z 719.846,A -85,B 0,C 180,E1 8988.84,E2 8988.84} C_VEL
LIN {X 0,Y 428.082,Z 724.797,A -85,B 0,C 180,E1 8991.899,E2 8991.899} C_VEL
LIN {X 0,Y 427.977,Z 725.984,A -85,B 0,C 180,E1 8993.933,E2 8993.933} C_VEL
LIN {X 0,Y 428.004,Z 724.669,A -85,B 0,C 180,E1 8996.973,E2 8996.973} C_VEL
LIN {X 0,Y 428.128,Z 718.615,A -85,B 0,C 180,E1 9000.51,E2 9000.51} C_VEL
LIN {X 0,Y 428.678,Z 707.129,A -85,B 0,C 180,E1 9004.042,E2 9004.042} C_VEL
LIN {X 0,Y 429.526,Z 690.23,A -85,B 0,C 180,E1 9007.321,E2 9007.321} C_VEL
LIN {X 0,Y 430.763,Z 667.735,A -85,B 0,C 180,E1 9010.241,E2 9010.241} C_VEL
LIN {X 0,Y 431.93,Z 641.596,A -85,B 0,C 180,E1 9012.489,E2 9012.489} C_VEL
LIN {X 0,Y 432.828,Z 613.115,A -85,B 0,C 180,E1 9014.002,E2 9014.002} C_VEL
LIN {X 0,Y 432.956,Z 578.744,A -85,B 0,C 180,E1 9014.893,E2 9014.893} C_VEL
LIN {X 0,Y 425.553,Z 549.53,A -85,B 0,C 180,E1 9015.811,E2 9015.811} C_VEL
LIN {X 0,Y 425.232,Z 549.53,A -85,B 0,C 180,E1 9022.982,E2 9022.982} C_VEL
LIN {X 0,Y 424.937,Z 549.53,A -85,B 0,C 180,E1 9029.818,E2 9029.818} C_VEL
LIN {X 0,Y 424.757,Z 549.53,A -85,B 0,C 180,E1 9037.16,E2 9037.16} C_VEL
LIN {X 0,Y 424.781,Z 549.53,A -85,B 0,C 180,E1 9042.458,E2 9042.458} C_VEL
LIN {X 0,Y 424.861,Z 549.53,A -85,B 0,C 180,E1 9048.242,E2 9048.242} C_VEL
LIN {X 0,Y 424.828,Z 549.53,A -85,B 0,C 180,E1 9055.362,E2 9055.362} C_VEL
LIN {X 0,Y 424.898,Z 549.53,A -85,B 0,C 180,E1 9055.945,E2 9055.945} C_VEL
LIN {X 0,Y 443.543,Z 593.492,A -85,B 0,C 180,E1 9059.206,E2 9059.206} C_VEL
LIN {X 0,Y 446.526,Z 604.265,A -85,B 0,C 180,E1 9059.961,E2 9059.961} C_VEL
LIN {X 0,Y 443.285,Z 639.528,A -85,B 0,C 180,E1 9061.888,E2 9061.888} C_VEL
LIN {X 0,Y 439.282,Z 673.078,A -85,B 0,C 180,E1 9064.568,E2 9064.568} C_VEL
LIN {X 0,Y 435.277,Z 702.49,A -85,B 0,C 180,E1 9067.849,E2 9067.849} C_VEL
LIN {X 0,Y 431.564,Z 729.194,A -85,B 0,C 180,E1 9071.92,E2 9071.92} C_VEL
LIN {X 0,Y 428.895,Z 749.792,A -85,B 0,C 180,E1 9076.26,E2 9076.26} C_VEL
LIN {X 0,Y 427.321,Z 765.477,A -85,B 0,C 180,E1 9080.958,E2 9080.958} C_VEL
LIN {X 0,Y 426.655,Z 775.845,A -85,B 0,C 180,E1 9085.944,E2 9085.944} C_VEL
LIN {X 0,Y 426.533,Z 780.222,A -85,B 0,C 180,E1 9090,E2 9090} C_VEL
LIN {X 0,Y 426.357,Z 781.009,A -85,B 0,C 180,E1 9094.06,E2 9094.06} C_VEL
LIN {X 0,Y 426.516,Z 777.063,A -85,B 0,C 180,E1 9099.162,E2 9099.162} C_VEL
LIN {X 0,Y 427.08,Z 768.596,A -85,B 0,C 180,E1 9103.726,E2 9103.726} C_VEL
LIN {X 0,Y 428.472,Z 754.313,A -85,B 0,C 180,E1 9108.482,E2 9108.482} C_VEL
LIN {X 0,Y 430.859,Z 735.041,A -85,B 0,C 180,E1 9112.935,E2 9112.935} C_VEL
LIN {X 0,Y 434.377,Z 709.963,A -85,B 0,C 180,E1 9117.101,E2 9117.101} C_VEL
LIN {X 0,Y 438.549,Z 680.246,A -85,B 0,C 180,E1 9120.713,E2 9120.713} C_VEL
LIN {X 0,Y 442.778,Z 646.865,A -85,B 0,C 180,E1 9123.612,E2 9123.612} C_VEL
LIN {X 0,Y 446.419,Z 610.511,A -85,B 0,C 180,E1 9125.772,E2 9125.772} C_VEL
LIN {X 0,Y 446.37,Z 600.787,A -85,B 0,C 180,E1 9126.278,E2 9126.278} C_VEL
LIN {X 0,Y 435.736,Z 572.239,A -85,B 0,C 180,E1 9128.419,E2 9128.419} C_VEL
LIN {X 0,Y 424.914,Z 549.53,A -85,B 0,C 180,E1 9130.36,E2 9130.36} C_VEL
LIN {X 0,Y 424.832,Z 549.53,A -85,B 0,C 180,E1 9137.548,E2 9137.548} C_VEL
LIN {X 0,Y 424.999,Z 549.53,A -85,B 0,C 180,E1 9142.865,E2 9142.865} C_VEL
LIN {X 0,Y 425.071,Z 549.53,A -85,B 0,C 180,E1 9148.442,E2 9148.442} C_VEL
LIN {X 0,Y 425.027,Z 549.53,A -85,B 0,C 180,E1 9154.778,E2 9154.778} C_VEL
LIN {X 0,Y 425.232,Z 549.53,A -85,B 0,C 180,E1 9157.865,E2 9157.865} C_VEL
LIN {X 0,Y 431.704,Z 580.032,A -85,B 0,C 180,E1 9158.69,E2 9158.69} C_VEL
LIN {X 0,Y 431.445,Z 628.891,A -85,B 0,C 180,E1 9159.74,E2 9159.74} C_VEL
LIN {X 0,Y 430.88,Z 655.474,A -85,B 0,C 180,E1 9161.118,E2 9161.118} C_VEL
LIN {X 0,Y 430.042,Z 678.862,A -85,B 0,C 180,E1 9163.168,E2 9163.168} C_VEL
LIN {X 0,Y 429.099,Z 698.024,A -85,B 0,C 180,E1 9165.744,E2 9165.744} C_VEL
LIN {X 0,Y 428.508,Z 712.852,A -85,B 0,C 180,E1 9168.827,E2 9168.827} C_VEL
LIN {X 0,Y 428.084,Z 721.727,A -85,B 0,C 180,E1 9171.889,E2 9171.889} C_VEL
LIN {X 0,Y 428.022,Z 725.004,A -85,B 0,C 180,E1 9173.924,E2 9173.924} C_VEL
LIN {X 0,Y 428.043,Z 726.374,A -85,B 0,C 180,E1 9175.952,E2 9175.952} C_VEL
LIN {X 0,Y 428.206,Z 724.869,A -85,B 0,C 180,E1 9178.986,E2 9178.986} C_VEL
LIN {X 0,Y 428.797,Z 717.46,A -85,B 0,C 180,E1 9182.517,E2 9182.517} C_VEL
LIN {X 0,Y 429.701,Z 704.055,A -85,B 0,C 180,E1 9185.79,E2 9185.79} C_VEL
LIN {X 0,Y 430.705,Z 685.528,A -85,B 0,C 180,E1 9188.559,E2 9188.559} C_VEL
LIN {X 0,Y 431.561,Z 663.39,A -85,B 0,C 180,E1 9190.664,E2 9190.664} C_VEL
LIN {X 0,Y 432.022,Z 638.462,A -85,B 0,C 180,E1 9192.093,E2 9192.093} C_VEL
LIN {X 0,Y 432.017,Z 605.449,A -85,B 0,C 180,E1 9192.957,E2 9192.957} C_VEL
LIN {X 0,Y 431.549,Z 572.274,A -85,B 0,C 180,E1 9193.631,E2 9193.631} C_VEL
LIN {X 0,Y 425.461,Z 549.53,A -85,B 0,C 180,E1 9194.502,E2 9194.502} C_VEL
LIN {X 0,Y 425.219,Z 549.53,A -85,B 0,C 180,E1 9200.781,E2 9200.781} C_VEL
LIN {X 0,Y 424.97,Z 549.53,A -85,B 0,C 180,E1 9207.486,E2 9207.486} C_VEL
LIN {X 0,Y 424.821,Z 549.53,A -85,B 0,C 180,E1 9214.629,E2 9214.629} C_VEL
LIN {X 0,Y 424.864,Z 549.53,A -85,B 0,C 180,E1 9219.735,E2 9219.735} C_VEL
LIN {X 0,Y 424.899,Z 550.07,A -85,B 0,C 180,E1 9226.005,E2 9226.005} C_VEL
LIN {X 0,Y 433.06,Z 565.463,A -85,B 0,C 180,E1 9227.314,E2 9227.314} C_VEL
LIN {X 0,Y 441.779,Z 584.143,A -85,B 0,C 180,E1 9228.712,E2 9228.712} C_VEL
LIN {X 0,Y 453.092,Z 613.261,A -85,B 0,C 180,E1 9230.715,E2 9230.715} C_VEL
LIN {X 0,Y 454,Z 616.98,A -85,B 0,C 180,E1 9230.933,E2 9230.933} C_VEL
LIN {X 0,Y 449.877,Z 661.559,A -85,B 0,C 180,E1 9232.675,E2 9232.675} C_VEL
LIN {X 0,Y 446.703,Z 690.803,A -85,B 0,C 180,E1 9234.34,E2 9234.34} C_VEL
LIN {X 0,Y 441.205,Z 706.365,A -85,B 0,C 180,E1 9235.159,E2 9235.159} C_VEL
LIN {X 0,Y 435.909,Z 721.251,A -85,B 0,C 180,E1 9236.106,E2 9236.106} C_VEL
LIN {X 0,Y 431.235,Z 753.12,A -85,B 0,C 180,E1 9239.256,E2 9239.256} C_VEL
LIN {X 0,Y 426.632,Z 782.447,A -85,B 0,C 180,E1 9243.19,E2 9243.19} C_VEL
LIN {X 0,Y 422.694,Z 808.809,A -85,B 0,C 180,E1 9247.989,E2 9247.989} C_VEL
LIN {X 0,Y 420.17,Z 828.663,A -85,B 0,C 180,E1 9252.916,E2 9252.916} C_VEL
LIN {X 0,Y 418.864,Z 843.289,A -85,B 0,C 180,E1 9258.043,E2 9258.043} C_VEL
LIN {X 0,Y 418.423,Z 851.589,A -85,B 0,C 180,E1 9262.472,E2 9262.472} C_VEL
LIN {X 0,Y 418.221,Z 856.591,A -85,B 0,C 180,E1 9267.932,E2 9267.932} C_VEL
LIN {X 0,Y 418.279,Z 856.598,A -85,B 0,C 180,E1 9272.067,E2 9272.067} C_VEL
LIN {X 0,Y 418.428,Z 851.583,A -85,B 0,C 180,E1 9277.537,E2 9277.537} C_VEL
LIN {X 0,Y 419.099,Z 840.629,A -85,B 0,C 180,E1 9283.062,E2 9283.062} C_VEL
LIN {X 0,Y 420.656,Z 824.538,A -85,B 0,C 180,E1 9288.255,E2 9288.255} C_VEL
LIN {X 0,Y 423.415,Z 803.682,A -85,B 0,C 180,E1 9293.083,E2 9293.083} C_VEL
LIN {X 0,Y 427.444,Z 777.56,A -85,B 0,C 180,E1 9297.57,E2 9297.57} C_VEL
LIN {X 0,Y 432.097,Z 747.861,A -85,B 0,C 180,E1 9301.359,E2 9301.359} C_VEL
LIN {X 0,Y 437.124,Z 712.792,A -85,B 0,C 180,E1 9304.606,E2 9304.606} C_VEL
LIN {X 0,Y 442.001,Z 672.855,A -85,B 0,C 180,E1 9307.267,E2 9307.267} C_VEL
LIN {X 0,Y 446.206,Z 631.748,A -85,B 0,C 180,E1 9309.129,E2 9309.129} C_VEL
LIN {X 0,Y 447.046,Z 616.221,A -85,B 0,C 180,E1 9309.687,E2 9309.687} C_VEL
LIN {X 0,Y 429.108,Z 573.372,A -85,B 0,C 180,E1 9312.719,E2 9312.719} C_VEL
LIN {X 0,Y 417.15,Z 551.057,A -85,B 0,C 180,E1 9314.562,E2 9314.562} C_VEL
LIN {X 0,Y 417.001,Z 549.53,A -85,B 0,C 180,E1 9314.758,E2 9314.758} C_VEL
LIN {X 0,Y 417.006,Z 549.53,A -85,B 0,C 180,E1 9322.041,E2 9322.041} C_VEL
LIN {X 0,Y 417.011,Z 549.53,A -85,B 0,C 180,E1 9329.567,E2 9329.567} C_VEL
LIN {X 0,Y 417.244,Z 549.53,A -85,B 0,C 180,E1 9333.349,E2 9333.349} C_VEL
LIN {X 0,Y 425.745,Z 580.127,A -85,B 0,C 180,E1 9334.547,E2 9334.547} C_VEL
LIN {X 0,Y 425.955,Z 620.621,A -85,B 0,C 180,E1 9335.566,E2 9335.566} C_VEL
LIN {X 0,Y 425.347,Z 649.578,A -85,B 0,C 180,E1 9337.112,E2 9337.112} C_VEL
LIN {X 0,Y 424.245,Z 674.884,A -85,B 0,C 180,E1 9339.355,E2 9339.355} C_VEL
LIN {X 0,Y 422.964,Z 695.202,A -85,B 0,C 180,E1 9342.083,E2 9342.083} C_VEL
LIN {X 0,Y 421.696,Z 711.765,A -85,B 0,C 180,E1 9345.498,E2 9345.498} C_VEL
LIN {X 0,Y 420.867,Z 722.251,A -85,B 0,C 180,E1 9349.155,E2 9349.155} C_VEL
LIN {X 0,Y 420.346,Z 726.163,A -85,B 0,C 180,E1 9351.749,E2 9351.749} C_VEL
LIN {X 0,Y 420.205,Z 727.367,A -85,B 0,C 180,E1 9353.82,E2 9353.82} C_VEL
LIN {X 0,Y 420.218,Z 726.08,A -85,B 0,C 180,E1 9356.917,E2 9356.917} C_VEL
LIN {X 0,Y 420.34,Z 719.988,A -85,B 0,C 180,E1 9360.519,E2 9360.519} C_VEL
LIN {X 0,Y 420.928,Z 708.446,A -85,B 0,C 180,E1 9364.116,E2 9364.116} C_VEL
LIN {X 0,Y 421.781,Z 691.458,A -85,B 0,C 180,E1 9367.457,E2 9367.457} C_VEL
LIN {X 0,Y 423.012,Z 670.255,A -85,B 0,C 180,E1 9370.279,E2 9370.279} C_VEL
LIN {X 0,Y 424.245,Z 644.37,A -85,B 0,C 180,E1 9372.588,E2 9372.588} C_VEL
LIN {X 0,Y 425.155,Z 615.594,A -85,B 0,C 180,E1 9374.194,E2 9374.194} C_VEL
LIN {X 0,Y 425.574,Z 581.345,A -85,B 0,C 180,E1 9375.124,E2 9375.124} C_VEL
LIN {X 0,Y 417.635,Z 549.53,A -85,B 0,C 180,E1 9376.138,E2 9376.138} C_VEL
LIN {X 0,Y 417.258,Z 549.53,A -85,B 0,C 180,E1 9383.447,E2 9383.447} C_VEL
LIN {X 0,Y 417.022,Z 549.53,A -85,B 0,C 180,E1 9390.443,E2 9390.443} C_VEL
LIN {X 0,Y 416.853,Z 549.53,A -85,B 0,C 180,E1 9397.204,E2 9397.204} C_VEL
LIN {X 0,Y 416.806,Z 549.53,A -85,B 0,C 180,E1 9403.601,E2 9403.601} C_VEL
LIN {X 0,Y 416.895,Z 549.53,A -85,B 0,C 180,E1 9409.483,E2 9409.483} C_VEL
LIN {X 0,Y 416.918,Z 549.53,A -85,B 0,C 180,E1 9415.111,E2 9415.111} C_VEL
LIN {X 0,Y 435.995,Z 593.557,A -85,B 0,C 180,E1 9418.543,E2 9418.543} C_VEL
LIN {X 0,Y 439.651,Z 607.193,A -85,B 0,C 180,E1 9419.524,E2 9419.524} C_VEL
LIN {X 0,Y 436.144,Z 643.143,A -85,B 0,C 180,E1 9421.574,E2 9421.574} C_VEL
LIN {X 0,Y 431.849,Z 676.59,A -85,B 0,C 180,E1 9424.376,E2 9424.376} C_VEL
LIN {X 0,Y 427.735,Z 705.312,A -85,B 0,C 180,E1 9427.711,E2 9427.711} C_VEL
LIN {X 0,Y 423.843,Z 731.381,A -85,B 0,C 180,E1 9431.847,E2 9431.847} C_VEL
LIN {X 0,Y 421.105,Z 751.588,A -85,B 0,C 180,E1 9436.265,E2 9436.265} C_VEL
LIN {X 0,Y 419.569,Z 765.931,A -85,B 0,C 180,E1 9440.685,E2 9440.685} C_VEL
LIN {X 0,Y 418.897,Z 774.943,A -85,B 0,C 180,E1 9444.833,E2 9444.833} C_VEL
LIN {X 0,Y 418.663,Z 780.949,A -85,B 0,C 180,E1 9450,E2 9450} C_VEL
LIN {X 0,Y 418.5,Z 781.706,A -85,B 0,C 180,E1 9454.136,E2 9454.136} C_VEL
LIN {X 0,Y 418.664,Z 777.654,A -85,B 0,C 180,E1 9459.336,E2 9459.336} C_VEL
LIN {X 0,Y 419.421,Z 767.61,A -85,B 0,C 180,E1 9464.589,E2 9464.589} C_VEL
LIN {X 0,Y 421.124,Z 751.813,A -85,B 0,C 180,E1 9469.632,E2 9469.632} C_VEL
LIN {X 0,Y 424.041,Z 730.484,A -85,B 0,C 180,E1 9474.304,E2 9474.304} C_VEL
LIN {X 0,Y 428.141,Z 703.887,A -85,B 0,C 180,E1 9478.481,E2 9478.481} C_VEL
LIN {X 0,Y 432.705,Z 673.206,A -85,B 0,C 180,E1 9481.983,E2 9481.983} C_VEL
LIN {X 0,Y 436.855,Z 641.086,A -85,B 0,C 180,E1 9484.601,E2 9484.601} C_VEL
LIN {X 0,Y 440.014,Z 604.16,A -85,B 0,C 180,E1 9486.705,E2 9486.705} C_VEL
LIN {X 0,Y 429.997,Z 576.487,A -85,B 0,C 180,E1 9488.868,E2 9488.868} C_VEL
LIN {X 0,Y 417.045,Z 550.677,A -85,B 0,C 180,E1 9491.202,E2 9491.202} C_VEL
LIN {X 0,Y 416.948,Z 549.53,A -85,B 0,C 180,E1 9491.463,E2 9491.463} C_VEL
LIN {X 0,Y 416.835,Z 549.53,A -85,B 0,C 180,E1 9496.534,E2 9496.534} C_VEL
LIN {X 0,Y 417.105,Z 549.53,A -85,B 0,C 180,E1 9502.751,E2 9502.751} C_VEL
LIN {X 0,Y 417.104,Z 549.53,A -85,B 0,C 180,E1 9509.563,E2 9509.563} C_VEL
LIN {X 0,Y 417.262,Z 549.53,A -85,B 0,C 180,E1 9517.295,E2 9517.295} C_VEL
LIN {X 0,Y 417.297,Z 549.53,A -85,B 0,C 180,E1 9517.555,E2 9517.555} C_VEL
LIN {X 0,Y 424.012,Z 579.86,A -85,B 0,C 180,E1 9518.414,E2 9518.414} C_VEL
LIN {X 0,Y 423.775,Z 630.237,A -85,B 0,C 180,E1 9519.522,E2 9519.522} C_VEL
LIN {X 0,Y 423.147,Z 657.411,A -85,B 0,C 180,E1 9520.97,E2 9520.97} C_VEL
LIN {X 0,Y 422.309,Z 681.086,A -85,B 0,C 180,E1 9523.117,E2 9523.117} C_VEL
LIN {X 0,Y 421.294,Z 699.946,A -85,B 0,C 180,E1 9525.739,E2 9525.739} C_VEL
LIN {X 0,Y 420.769,Z 713.606,A -85,B 0,C 180,E1 9528.619,E2 9528.619} C_VEL
LIN {X 0,Y 420.331,Z 722.756,A -85,B 0,C 180,E1 9531.739,E2 9531.739} C_VEL
LIN {X 0,Y 420.244,Z 726.191,A -85,B 0,C 180,E1 9533.811,E2 9533.811} C_VEL
LIN {X 0,Y 420.269,Z 727.67,A -85,B 0,C 180,E1 9535.877,E2 9535.877} C_VEL
LIN {X 0,Y 420.445,Z 726.346,A -85,B 0,C 180,E1 9538.967,E2 9538.967} C_VEL
LIN {X 0,Y 421.09,Z 719.122,A -85,B 0,C 180,E1 9542.563,E2 9542.563} C_VEL
LIN {X 0,Y 422.037,Z 705.887,A -85,B 0,C 180,E1 9545.896,E2 9545.896} C_VEL
LIN {X 0,Y 423.105,Z 687.568,A -85,B 0,C 180,E1 9548.714,E2 9548.714} C_VEL
LIN {X 0,Y 424.051,Z 665.009,A -85,B 0,C 180,E1 9550.915,E2 9550.915} C_VEL
LIN {X 0,Y 424.517,Z 639.847,A -85,B 0,C 180,E1 9552.384,E2 9552.384} C_VEL
LIN {X 0,Y 424.539,Z 606.062,A -85,B 0,C 180,E1 9553.277,E2 9553.277} C_VEL
LIN {X 0,Y 424.059,Z 573.153,A -85,B 0,C 180,E1 9553.982,E2 9553.982} C_VEL
LIN {X 0,Y 417.542,Z 549.53,A -85,B 0,C 180,E1 9554.917,E2 9554.917} C_VEL
LIN {X 0,Y 417.293,Z 549.53,A -85,B 0,C 180,E1 9561.195,E2 9561.195} C_VEL
LIN {X 0,Y 416.977,Z 549.53,A -85,B 0,C 180,E1 9568.059,E2 9568.059} C_VEL
LIN {X 0,Y 416.897,Z 549.53,A -85,B 0,C 180,E1 9575.385,E2 9575.385} C_VEL
LIN {X 0,Y 416.931,Z 549.53,A -85,B 0,C 180,E1 9580.647,E2 9580.647} C_VEL
LIN {X 0,Y 417.01,Z 550.254,A -85,B 0,C 180,E1 9585.015,E2 9585.015} C_VEL
LIN {X 0,Y 434.822,Z 584.55,A -85,B 0,C 180,E1 9587.984,E2 9587.984} C_VEL
LIN {X 0,Y 446.822,Z 616.735,A -85,B 0,C 180,E1 9590.268,E2 9590.268} C_VEL
LIN {X 0,Y 444.986,Z 645.224,A -85,B 0,C 180,E1 9591.372,E2 9591.372} C_VEL
LIN {X 0,Y 440.464,Z 686.334,A -85,B 0,C 180,E1 9593.529,E2 9593.529} C_VEL
LIN {X 0,Y 435.909,Z 721.251,A -85,B 0,C 180,E1 9596.106,E2 9596.106} C_VEL
LIN {X 0,Y 430.446,Z 735.79,A -85,B 0,C 180,E1 9597.179,E2 9597.179} C_VEL
LIN {X 0,Y 424.588,Z 749.654,A -85,B 0,C 180,E1 9598.389,E2 9598.389} C_VEL
LIN {X 0,Y 419.616,Z 780.095,A -85,B 0,C 180,E1 9602.415,E2 9602.415} C_VEL
LIN {X 0,Y 415.368,Z 806.151,A -85,B 0,C 180,E1 9607.126,E2 9607.126} C_VEL
LIN {X 0,Y 412.641,Z 825.815,A -85,B 0,C 180,E1 9611.941,E2 9611.941} C_VEL
LIN {X 0,Y 411.084,Z 841.387,A -85,B 0,C 180,E1 9617.275,E2 9617.275} C_VEL
LIN {X 0,Y 410.554,Z 851.042,A -85,B 0,C 180,E1 9622.437,E2 9622.437} C_VEL
LIN {X 0,Y 410.344,Z 855.883,A -85,B 0,C 180,E1 9627.892,E2 9627.892} C_VEL
LIN {X 0,Y 410.401,Z 855.893,A -85,B 0,C 180,E1 9632.107,E2 9632.107} C_VEL
LIN {X 0,Y 410.561,Z 851.046,A -85,B 0,C 180,E1 9637.573,E2 9637.573} C_VEL
LIN {X 0,Y 411.116,Z 841.431,A -85,B 0,C 180,E1 9642.724,E2 9642.724} C_VEL
LIN {X 0,Y 412.735,Z 825.741,A -85,B 0,C 180,E1 9648.099,E2 9648.099} C_VEL
LIN {X 0,Y 415.617,Z 804.663,A -85,B 0,C 180,E1 9653.203,E2 9653.203} C_VEL
LIN {X 0,Y 419.889,Z 778.479,A -85,B 0,C 180,E1 9657.856,E2 9657.856} C_VEL
LIN {X 0,Y 424.663,Z 749.437,A -85,B 0,C 180,E1 9661.656,E2 9661.656} C_VEL
LIN {X 0,Y 429.826,Z 714.835,A -85,B 0,C 180,E1 9664.942,E2 9664.942} C_VEL
LIN {X 0,Y 434.971,Z 674.739,A -85,B 0,C 180,E1 9667.695,E2 9667.695} C_VEL
LIN {X 0,Y 439.489,Z 633.054,A -85,B 0,C 180,E1 9669.65,E2 9669.65} C_VEL
LIN {X 0,Y 440.164,Z 618.509,A -85,B 0,C 180,E1 9670.211,E2 9670.211} C_VEL
LIN {X 0,Y 423.925,Z 578.371,A -85,B 0,C 180,E1 9673.153,E2 9673.153} C_VEL
LIN {X 0,Y 409.204,Z 550.93,A -85,B 0,C 180,E1 9675.526,E2 9675.526} C_VEL
LIN {X 0,Y 409.072,Z 549.53,A -85,B 0,C 180,E1 9675.645,E2 9675.645} C_VEL
LIN {X 0,Y 408.992,Z 549.53,A -85,B 0,C 180,E1 9681.16,E2 9681.16} C_VEL
LIN {X 0,Y 408.991,Z 549.53,A -85,B 0,C 180,E1 9688.07,E2 9688.07} C_VEL
LIN {X 0,Y 409.255,Z 549.53,A -85,B 0,C 180,E1 9692.807,E2 9692.807} C_VEL
LIN {X 0,Y 418.423,Z 581.224,A -85,B 0,C 180,E1 9694.159,E2 9694.159} C_VEL
LIN {X 0,Y 418.584,Z 622.733,A -85,B 0,C 180,E1 9695.24,E2 9695.24} C_VEL
LIN {X 0,Y 417.925,Z 651.762,A -85,B 0,C 180,E1 9696.839,E2 9696.839} C_VEL
LIN {X 0,Y 416.804,Z 676.269,A -85,B 0,C 180,E1 9699.051,E2 9699.051} C_VEL
LIN {X 0,Y 415.467,Z 696.194,A -85,B 0,C 180,E1 9701.749,E2 9701.749} C_VEL
LIN {X 0,Y 414.259,Z 711.032,A -85,B 0,C 180,E1 9704.726,E2 9704.726} C_VEL
LIN {X 0,Y 413.277,Z 722.446,A -85,B 0,C 180,E1 9708.42,E2 9708.42} C_VEL
LIN {X 0,Y 412.636,Z 727.547,A -85,B 0,C 180,E1 9711.593,E2 9711.593} C_VEL
LIN {X 0,Y 412.441,Z 728.767,A -85,B 0,C 180,E1 9713.703,E2 9713.703} C_VEL
LIN {X 0,Y 412.432,Z 727.486,A -85,B 0,C 180,E1 9716.859,E2 9716.859} C_VEL
LIN {X 0,Y 412.579,Z 721.372,A -85,B 0,C 180,E1 9720.529,E2 9720.529} C_VEL
LIN {X 0,Y 413.155,Z 709.767,A -85,B 0,C 180,E1 9724.194,E2 9724.194} C_VEL
LIN {X 0,Y 414.043,Z 692.705,A -85,B 0,C 180,E1 9727.597,E2 9727.597} C_VEL
LIN {X 0,Y 415.321,Z 671.39,A -85,B 0,C 180,E1 9730.472,E2 9730.472} C_VEL
LIN {X 0,Y 416.616,Z 645.376,A -85,B 0,C 180,E1 9732.823,E2 9732.823} C_VEL
LIN {X 0,Y 417.55,Z 616.411,A -85,B 0,C 180,E1 9734.458,E2 9734.458} C_VEL
LIN {X 0,Y 417.824,Z 581.412,A -85,B 0,C 180,E1 9735.422,E2 9735.422} C_VEL
LIN {X 0,Y 409.701,Z 549.53,A -85,B 0,C 180,E1 9736.489,E2 9736.489} C_VEL
LIN {X 0,Y 409.314,Z 549.53,A -85,B 0,C 180,E1 9743.93,E2 9743.93} C_VEL
LIN {X 0,Y 409.013,Z 549.53,A -85,B 0,C 180,E1 9751.105,E2 9751.105} C_VEL
LIN {X 0,Y 408.916,Z 549.53,A -85,B 0,C 180,E1 9756.195,E2 9756.195} C_VEL
LIN {X 0,Y 408.808,Z 549.53,A -85,B 0,C 180,E1 9762.411,E2 9762.411} C_VEL
LIN {X 0,Y 408.874,Z 549.53,A -85,B 0,C 180,E1 9768.365,E2 9768.365} C_VEL
LIN {X 0,Y 408.976,Z 549.53,A -85,B 0,C 180,E1 9774.216,E2 9774.216} C_VEL
LIN {X 0,Y 428.406,Z 593.402,A -85,B 0,C 180,E1 9777.837,E2 9777.837} C_VEL
LIN {X 0,Y 432.956,Z 608.567,A -85,B 0,C 180,E1 9779.001,E2 9779.001} C_VEL
LIN {X 0,Y 429.305,Z 644.163,A -85,B 0,C 180,E1 9781.072,E2 9781.072} C_VEL
LIN {X 0,Y 424.792,Z 677.574,A -85,B 0,C 180,E1 9783.919,E2 9783.919} C_VEL
LIN {X 0,Y 420.46,Z 706.204,A -85,B 0,C 180,E1 9787.304,E2 9787.304} C_VEL
LIN {X 0,Y 416.349,Z 732.214,A -85,B 0,C 180,E1 9791.509,E2 9791.509} C_VEL
LIN {X 0,Y 413.436,Z 752.377,A -85,B 0,C 180,E1 9796.006,E2 9796.006} C_VEL
LIN {X 0,Y 411.652,Z 768.017,A -85,B 0,C 180,E1 9801.037,E2 9801.037} C_VEL
LIN {X 0,Y 410.959,Z 777.336,A -85,B 0,C 180,E1 9805.788,E2 9805.788} C_VEL
LIN {X 0,Y 410.814,Z 781.673,A -85,B 0,C 180,E1 9810,E2 9810} C_VEL
LIN {X 0,Y 410.643,Z 782.404,A -85,B 0,C 180,E1 9814.216,E2 9814.216} C_VEL
LIN {X 0,Y 410.845,Z 778.265,A -85,B 0,C 180,E1 9819.515,E2 9819.515} C_VEL
LIN {X 0,Y 411.558,Z 769.346,A -85,B 0,C 180,E1 9824.373,E2 9824.373} C_VEL
LIN {X 0,Y 413.223,Z 755.224,A -85,B 0,C 180,E1 9829.19,E2 9829.19} C_VEL
LIN {X 0,Y 416.101,Z 734.992,A -85,B 0,C 180,E1 9833.961,E2 9833.961} C_VEL
LIN {X 0,Y 420.087,Z 710.437,A -85,B 0,C 180,E1 9838.128,E2 9838.128} C_VEL
LIN {X 0,Y 424.741,Z 681.182,A -85,B 0,C 180,E1 9841.761,E2 9841.761} C_VEL
LIN {X 0,Y 429.355,Z 648.55,A -85,B 0,C 180,E1 9844.68,E2 9844.68} C_VEL
LIN {X 0,Y 433.334,Z 612.521,A -85,B 0,C 180,E1 9846.887,E2 9846.887} C_VEL
LIN {X 0,Y 432.79,Z 604.209,A -85,B 0,C 180,E1 9847.401,E2 9847.401} C_VEL
LIN {X 0,Y 423.336,Z 578.613,A -85,B 0,C 180,E1 9849.502,E2 9849.502} C_VEL
LIN {X 0,Y 409.122,Z 550.428,A -85,B 0,C 180,E1 9852.195,E2 9852.195} C_VEL
LIN {X 0,Y 409.059,Z 549.53,A -85,B 0,C 180,E1 9852.448,E2 9852.448} C_VEL
LIN {X 0,Y 408.883,Z 549.53,A -85,B 0,C 180,E1 9858.364,E2 9858.364} C_VEL
LIN {X 0,Y 409.174,Z 549.53,A -85,B 0,C 180,E1 9864.237,E2 9864.237} C_VEL
LIN {X 0,Y 409.127,Z 549.53,A -85,B 0,C 180,E1 9871.342,E2 9871.342} C_VEL
LIN {X 0,Y 409.358,Z 549.53,A -85,B 0,C 180,E1 9877.234,E2 9877.234} C_VEL
LIN {X 0,Y 416.458,Z 582.216,A -85,B 0,C 180,E1 9878.181,E2 9878.181} C_VEL
LIN {X 0,Y 416.14,Z 631.388,A -85,B 0,C 180,E1 9879.29,E2 9879.29} C_VEL
LIN {X 0,Y 415.473,Z 658.28,A -85,B 0,C 180,E1 9880.742,E2 9880.742} C_VEL
LIN {X 0,Y 414.613,Z 682.13,A -85,B 0,C 180,E1 9882.931,E2 9882.931} C_VEL
LIN {X 0,Y 413.517,Z 701.863,A -85,B 0,C 180,E1 9885.735,E2 9885.735} C_VEL
LIN {X 0,Y 412.887,Z 716.278,A -85,B 0,C 180,E1 9888.933,E2 9888.933} C_VEL
LIN {X 0,Y 412.47,Z 725.35,A -85,B 0,C 180,E1 9892.383,E2 9892.383} C_VEL
LIN {X 0,Y 412.5,Z 728.962,A -85,B 0,C 180,E1 9895.799,E2 9895.799} C_VEL
LIN {X 0,Y 412.676,Z 727.821,A -85,B 0,C 180,E1 9898.948,E2 9898.948} C_VEL
LIN {X 0,Y 413.355,Z 720.779,A -85,B 0,C 180,E1 9902.611,E2 9902.611} C_VEL
LIN {X 0,Y 414.331,Z 708.995,A -85,B 0,C 180,E1 9905.743,E2 9905.743} C_VEL
LIN {X 0,Y 415.452,Z 691.649,A -85,B 0,C 180,E1 9908.612,E2 9908.612} C_VEL
LIN {X 0,Y 416.458,Z 669.846,A -85,B 0,C 180,E1 9910.914,E2 9910.914} C_VEL
LIN {X 0,Y 417.069,Z 644.649,A -85,B 0,C 180,E1 9912.533,E2 9912.533} C_VEL
LIN {X 0,Y 417.035,Z 615.494,A -85,B 0,C 180,E1 9913.445,E2 9913.445} C_VEL
LIN {X 0,Y 416.816,Z 575.22,A -85,B 0,C 180,E1 9914.307,E2 9914.307} C_VEL
LIN {X 0,Y 409.601,Z 549.53,A -85,B 0,C 180,E1 9915.366,E2 9915.366} C_VEL
LIN {X 0,Y 409.316,Z 549.53,A -85,B 0,C 180,E1 9921.628,E2 9921.628} C_VEL
LIN {X 0,Y 409.038,Z 549.53,A -85,B 0,C 180,E1 9928.654,E2 9928.654} C_VEL
LIN {X 0,Y 409.01,Z 549.53,A -85,B 0,C 180,E1 9936.173,E2 9936.173} C_VEL
LIN {X 0,Y 408.999,Z 549.53,A -85,B 0,C 180,E1 9943.681,E2 9943.681} C_VEL
LIN {X 0,Y 409.04,Z 550.076,A -85,B 0,C 180,E1 9943.948,E2 9943.948} C_VEL
LIN {X 0,Y 414.368,Z 560.303,A -85,B 0,C 180,E1 9944.91,E2 9944.91} C_VEL
LIN {X 0,Y 429.077,Z 588.278,A -85,B 0,C 180,E1 9947.466,E2 9947.466} C_VEL
LIN {X 0,Y 440.725,Z 622.416,A -85,B 0,C 180,E1 9949.917,E2 9949.917} C_VEL
LIN {X 0,Y 436.028,Z 666.623,A -85,B 0,C 180,E1 9951.825,E2 9951.825} C_VEL
LIN {X 0,Y 430.681,Z 708.221,A -85,B 0,C 180,E1 9954.522,E2 9954.522} C_VEL
LIN {X 0,Y 425.191,Z 745.764,A -85,B 0,C 180,E1 9957.961,E2 9957.961} C_VEL
LIN {X 0,Y 424.588,Z 749.654,A -85,B 0,C 180,E1 9958.389,E2 9958.389} C_VEL
LIN {X 0,Y 418.799,Z 762.883,A -85,B 0,C 180,E1 9959.755,E2 9959.755} C_VEL
LIN {X 0,Y 413.08,Z 775.272,A -85,B 0,C 180,E1 9961.262,E2 9961.262} C_VEL
LIN {X 0,Y 408.537,Z 801.387,A -85,B 0,C 180,E1 9965.8,E2 9965.8} C_VEL
LIN {X 0,Y 405.206,Z 823.196,A -85,B 0,C 180,E1 9971.007,E2 9971.007} C_VEL
LIN {X 0,Y 403.343,Z 839.633,A -85,B 0,C 180,E1 9976.57,E2 9976.57} C_VEL
LIN {X 0,Y 402.709,Z 849.048,A -85,B 0,C 180,E1 9981.378,E2 9981.378} C_VEL
LIN {X 0,Y 402.461,Z 853.947,A -85,B 0,C 180,E1 9985.699,E2 9985.699} C_VEL
LIN {X 0,Y 402.543,Z 855.604,A -85,B 0,C 180,E1 9990,E2 9990} C_VEL
LIN {X 0,Y 402.512,Z 853.051,A -85,B 0,C 180,E1 9995.378,E2 9995.378} C_VEL
LIN {X 0,Y 402.887,Z 845.372,A -85,B 0,C 180,E1 10000.795,E2 10000.795} C_VEL
LIN {X 0,Y 404.151,Z 832.12,A -85,B 0,C 180,E1 10006.264,E2 10006.264} C_VEL
LIN {X 0,Y 406.763,Z 812.503,A -85,B 0,C 180,E1 10011.778,E2 10011.778} C_VEL
LIN {X 0,Y 410.615,Z 789.507,A -85,B 0,C 180,E1 10016.464,E2 10016.464} C_VEL
LIN {X 0,Y 415.524,Z 760.962,A -85,B 0,C 180,E1 10020.737,E2 10020.737} C_VEL
LIN {X 0,Y 420.658,Z 729.053,A -85,B 0,C 180,E1 10024.206,E2 10024.206} C_VEL
LIN {X 0,Y 426.276,Z 689.676,A -85,B 0,C 180,E1 10027.314,E2 10027.314} C_VEL
LIN {X 0,Y 431.365,Z 647.031,A -85,B 0,C 180,E1 10029.666,E2 10029.666} C_VEL
LIN {X 0,Y 433.654,Z 621.645,A -85,B 0,C 180,E1 10030.681,E2 10030.681} C_VEL
LIN {X 0,Y 418.333,Z 582.659,A -85,B 0,C 180,E1 10033.646,E2 10033.646} C_VEL
LIN {X 0,Y 401.204,Z 550.635,A -85,B 0,C 180,E1 10036.555,E2 10036.555} C_VEL
LIN {X 0,Y 401.1,Z 549.53,A -85,B 0,C 180,E1 10036.752,E2 10036.752} C_VEL
LIN {X 0,Y 401.038,Z 549.53,A -85,B 0,C 180,E1 10042.989,E2 10042.989} C_VEL
LIN {X 0,Y 401.077,Z 549.53,A -85,B 0,C 180,E1 10049.933,E2 10049.933} C_VEL
LIN {X 0,Y 401.275,Z 549.803,A -85,B 0,C 180,E1 10052.224,E2 10052.224} C_VEL
LIN {X 0,Y 410.379,Z 578.927,A -85,B 0,C 180,E1 10053.612,E2 10053.612} C_VEL
LIN {X 0,Y 411.294,Z 594.595,A -85,B 0,C 180,E1 10054.027,E2 10054.027} C_VEL
LIN {X 0,Y 411.186,Z 628.029,A -85,B 0,C 180,E1 10055.031,E2 10055.031} C_VEL
LIN {X 0,Y 410.491,Z 655.251,A -85,B 0,C 180,E1 10056.643,E2 10056.643} C_VEL
LIN {X 0,Y 409.272,Z 679.49,A -85,B 0,C 180,E1 10058.936,E2 10058.936} C_VEL
LIN {X 0,Y 407.907,Z 698.839,A -85,B 0,C 180,E1 10061.677,E2 10061.677} C_VEL
LIN {X 0,Y 406.512,Z 714.194,A -85,B 0,C 180,E1 10064.944,E2 10064.944} C_VEL
LIN {X 0,Y 405.519,Z 724.948,A -85,B 0,C 180,E1 10068.739,E2 10068.739} C_VEL
LIN {X 0,Y 404.928,Z 728.94,A -85,B 0,C 180,E1 10071.432,E2 10071.432} C_VEL
LIN {X 0,Y 404.677,Z 730.172,A -85,B 0,C 180,E1 10073.582,E2 10073.582} C_VEL
LIN {X 0,Y 404.648,Z 728.899,A -85,B 0,C 180,E1 10076.798,E2 10076.798} C_VEL
LIN {X 0,Y 404.811,Z 722.719,A -85,B 0,C 180,E1 10080.539,E2 10080.539} C_VEL
LIN {X 0,Y 405.385,Z 711.051,A -85,B 0,C 180,E1 10084.274,E2 10084.274} C_VEL
LIN {X 0,Y 406.302,Z 693.889,A -85,B 0,C 180,E1 10087.742,E2 10087.742} C_VEL
LIN {X 0,Y 407.635,Z 672.459,A -85,B 0,C 180,E1 10090.672,E2 10090.672} C_VEL
LIN {X 0,Y 408.98,Z 646.298,A -85,B 0,C 180,E1 10093.066,E2 10093.066} C_VEL
LIN {X 0,Y 409.943,Z 617.117,A -85,B 0,C 180,E1 10094.733,E2 10094.733} C_VEL
LIN {X 0,Y 410.052,Z 582.009,A -85,B 0,C 180,E1 10095.72,E2 10095.72} C_VEL
LIN {X 0,Y 401.742,Z 549.53,A -85,B 0,C 180,E1 10096.804,E2 10096.804} C_VEL
LIN {X 0,Y 401.462,Z 549.53,A -85,B 0,C 180,E1 10102.084,E2 10102.084} C_VEL
LIN {X 0,Y 401.119,Z 549.53,A -85,B 0,C 180,E1 10109.285,E2 10109.285} C_VEL
LIN {X 0,Y 401.026,Z 549.53,A -85,B 0,C 180,E1 10114.369,E2 10114.369} C_VEL
LIN {X 0,Y 400.864,Z 549.53,A -85,B 0,C 180,E1 10121.153,E2 10121.153} C_VEL
LIN {X 0,Y 400.945,Z 549.53,A -85,B 0,C 180,E1 10127.35,E2 10127.35} C_VEL
LIN {X 0,Y 401.002,Z 549.53,A -85,B 0,C 180,E1 10133.254,E2 10133.254} C_VEL
LIN {X 0,Y 421.34,Z 594.628,A -85,B 0,C 180,E1 10137.207,E2 10137.207} C_VEL
LIN {X 0,Y 426.175,Z 611.336,A -85,B 0,C 180,E1 10138.528,E2 10138.528} C_VEL
LIN {X 0,Y 422.278,Z 647.217,A -85,B 0,C 180,E1 10140.695,E2 10140.695} C_VEL
LIN {X 0,Y 417.578,Z 679.844,A -85,B 0,C 180,E1 10143.578,E2 10143.578} C_VEL
LIN {X 0,Y 412.912,Z 709.046,A -85,B 0,C 180,E1 10147.149,E2 10147.149} C_VEL
LIN {X 0,Y 408.659,Z 734.434,A -85,B 0,C 180,E1 10151.427,E2 10151.427} C_VEL
LIN {X 0,Y 405.635,Z 754.426,A -85,B 0,C 180,E1 10156.066,E2 10156.066} C_VEL
LIN {X 0,Y 403.882,Z 768.792,A -85,B 0,C 180,E1 10160.863,E2 10160.863} C_VEL
LIN {X 0,Y 403.136,Z 778.087,A -85,B 0,C 180,E1 10165.707,E2 10165.707} C_VEL
LIN {X 0,Y 402.944,Z 782.399,A -85,B 0,C 180,E1 10170,E2 10170} C_VEL
LIN {X 0,Y 402.784,Z 783.104,A -85,B 0,C 180,E1 10174.298,E2 10174.298} C_VEL
LIN {X 0,Y 403.001,Z 778.893,A -85,B 0,C 180,E1 10179.702,E2 10179.702} C_VEL
LIN {X 0,Y 403.79,Z 769.829,A -85,B 0,C 180,E1 10184.693,E2 10184.693} C_VEL
LIN {X 0,Y 405.58,Z 755.743,A -85,B 0,C 180,E1 10189.567,E2 10189.567} C_VEL
LIN {X 0,Y 408.658,Z 735.718,A -85,B 0,C 180,E1 10194.365,E2 10194.365} C_VEL
LIN {X 0,Y 413.066,Z 710.313,A -85,B 0,C 180,E1 10198.734,E2 10198.734} C_VEL
LIN {X 0,Y 417.924,Z 681.447,A -85,B 0,C 180,E1 10202.342,E2 10202.342} C_VEL
LIN {X 0,Y 422.8,Z 648.749,A -85,B 0,C 180,E1 10205.297,E2 10205.297} C_VEL
LIN {X 0,Y 426.92,Z 613.1,A -85,B 0,C 180,E1 10207.495,E2 10207.495} C_VEL
LIN {X 0,Y 425.329,Z 603.707,A -85,B 0,C 180,E1 10208.186,E2 10208.186} C_VEL
LIN {X 0,Y 415.519,Z 578.523,A -85,B 0,C 180,E1 10210.376,E2 10210.376} C_VEL
LIN {X 0,Y 401.123,Z 550.863,A -85,B 0,C 180,E1 10213.232,E2 10213.232} C_VEL
LIN {X 0,Y 400.99,Z 549.53,A -85,B 0,C 180,E1 10213.387,E2 10213.387} C_VEL
LIN {X 0,Y 401.026,Z 549.53,A -85,B 0,C 180,E1 10220.224,E2 10220.224} C_VEL
LIN {X 0,Y 401.231,Z 549.53,A -85,B 0,C 180,E1 10225.844,E2 10225.844} C_VEL
LIN {X 0,Y 401.177,Z 549.53,A -85,B 0,C 180,E1 10233.162,E2 10233.162} C_VEL
LIN {X 0,Y 401.416,Z 549.53,A -85,B 0,C 180,E1 10236.898,E2 10236.898} C_VEL
LIN {X 0,Y 408.801,Z 581.947,A -85,B 0,C 180,E1 10237.891,E2 10237.891} C_VEL
LIN {X 0,Y 408.496,Z 631.691,A -85,B 0,C 180,E1 10239.026,E2 10239.026} C_VEL
LIN {X 0,Y 407.845,Z 658.142,A -85,B 0,C 180,E1 10240.443,E2 10240.443} C_VEL
LIN {X 0,Y 406.955,Z 681.966,A -85,B 0,C 180,E1 10242.607,E2 10242.607} C_VEL
LIN {X 0,Y 405.84,Z 701.974,A -85,B 0,C 180,E1 10245.417,E2 10245.417} C_VEL
LIN {X 0,Y 405.131,Z 717.034,A -85,B 0,C 180,E1 10248.718,E2 10248.718} C_VEL
LIN {X 0,Y 404.68,Z 726.656,A -85,B 0,C 180,E1 10252.371,E2 10252.371} C_VEL
LIN {X 0,Y 404.722,Z 730.25,A -85,B 0,C 180,E1 10255.719,E2 10255.719} C_VEL
LIN {X 0,Y 404.917,Z 729.293,A -85,B 0,C 180,E1 10258.927,E2 10258.927} C_VEL
LIN {X 0,Y 405.629,Z 722.474,A -85,B 0,C 180,E1 10262.66,E2 10262.66} C_VEL
LIN {X 0,Y 406.674,Z 710.883,A -85,B 0,C 180,E1 10265.852,E2 10265.852} C_VEL
LIN {X 0,Y 407.877,Z 693.762,A -85,B 0,C 180,E1 10268.773,E2 10268.773} C_VEL
LIN {X 0,Y 408.913,Z 672.384,A -85,B 0,C 180,E1 10271.118,E2 10271.118} C_VEL
LIN {X 0,Y 409.595,Z 647.919,A -85,B 0,C 180,E1 10272.766,E2 10272.766} C_VEL
LIN {X 0,Y 409.61,Z 619.701,A -85,B 0,C 180,E1 10273.723,E2 10273.723} C_VEL
LIN {X 0,Y 409.32,Z 576.029,A -85,B 0,C 180,E1 10274.709,E2 10274.709} C_VEL
LIN {X 0,Y 401.695,Z 549.53,A -85,B 0,C 180,E1 10275.917,E2 10275.917} C_VEL
LIN {X 0,Y 401.373,Z 549.53,A -85,B 0,C 180,E1 10282.079,E2 10282.079} C_VEL
LIN {X 0,Y 401.04,Z 549.53,A -85,B 0,C 180,E1 10289.28,E2 10289.28} C_VEL
LIN {X 0,Y 401.032,Z 549.53,A -85,B 0,C 180,E1 10294.357,E2 10294.357} C_VEL
LIN {X 0,Y 400.97,Z 549.53,A -85,B 0,C 180,E1 10301.169,E2 10301.169} C_VEL
LIN {X 0,Y 401.088,Z 550.258,A -85,B 0,C 180,E1 10302.828,E2 10302.828} C_VEL
LIN {X 0,Y 407.151,Z 561.163,A -85,B 0,C 180,E1 10303.971,E2 10303.971} C_VEL
LIN {X 0,Y 423.496,Z 592.48,A -85,B 0,C 180,E1 10306.962,E2 10306.962} C_VEL
LIN {X 0,Y 434.138,Z 624.632,A -85,B 0,C 180,E1 10309.377,E2 10309.377} C_VEL
LIN {X 0,Y 429.263,Z 667.791,A -85,B 0,C 180,E1 10311.307,E2 10311.307} C_VEL
LIN {X 0,Y 423.754,Z 708.568,A -85,B 0,C 180,E1 10314.01,E2 10314.01} C_VEL
LIN {X 0,Y 418.042,Z 745.858,A -85,B 0,C 180,E1 10317.478,E2 10317.478} C_VEL
LIN {X 0,Y 413.08,Z 775.272,A -85,B 0,C 180,E1 10321.262,E2 10321.262} C_VEL
LIN {X 0,Y 407.232,Z 786.912,A -85,B 0,C 180,E1 10322.911,E2 10322.911} C_VEL
LIN {X 0,Y 401.587,Z 797.651,A -85,B 0,C 180,E1 10324.7,E2 10324.7} C_VEL
LIN {X 0,Y 397.971,Z 819.5,A -85,B 0,C 180,E1 10329.754,E2 10329.754} C_VEL
LIN {X 0,Y 395.831,Z 836.012,A -85,B 0,C 180,E1 10335.086,E2 10335.086} C_VEL
LIN {X 0,Y 394.969,Z 846.626,A -85,B 0,C 180,E1 10340.099,E2 10340.099} C_VEL
LIN {X 0,Y 394.584,Z 853.244,A -85,B 0,C 180,E1 10345.612,E2 10345.612} C_VEL
LIN {X 0,Y 394.695,Z 854.9,A -85,B 0,C 180,E1 10350,E2 10350} C_VEL
LIN {X 0,Y 394.602,Z 853.267,A -85,B 0,C 180,E1 10354.387,E2 10354.387} C_VEL
LIN {X 0,Y 394.903,Z 846.671,A -85,B 0,C 180,E1 10359.902,E2 10359.902} C_VEL
LIN {X 0,Y 395.99,Z 834.628,A -85,B 0,C 180,E1 10365.472,E2 10365.472} C_VEL
LIN {X 0,Y 398.213,Z 817.504,A -85,B 0,C 180,E1 10370.811,E2 10370.811} C_VEL
LIN {X 0,Y 401.989,Z 795.592,A -85,B 0,C 180,E1 10375.73,E2 10375.73} C_VEL
LIN {X 0,Y 406.763,Z 769.261,A -85,B 0,C 180,E1 10380.058,E2 10380.058} C_VEL
LIN {X 0,Y 412.033,Z 738.551,A -85,B 0,C 180,E1 10383.787,E2 10383.787} C_VEL
LIN {X 0,Y 417.878,Z 700.698,A -85,B 0,C 180,E1 10387.085,E2 10387.085} C_VEL
LIN {X 0,Y 423.455,Z 659.166,A -85,B 0,C 180,E1 10389.655,E2 10389.655} C_VEL
LIN {X 0,Y 426.841,Z 623.957,A -85,B 0,C 180,E1 10391.221,E2 10391.221} C_VEL
LIN {X 0,Y 412.792,Z 587.085,A -85,B 0,C 180,E1 10394.126,E2 10394.126} C_VEL
LIN {X 0,Y 393.162,Z 550.336,A -85,B 0,C 180,E1 10397.648,E2 10397.648} C_VEL
LIN {X 0,Y 393.089,Z 549.53,A -85,B 0,C 180,E1 10403.73,E2 10403.73} C_VEL
LIN {X 0,Y 393.176,Z 549.53,A -85,B 0,C 180,E1 10410.076,E2 10410.076} C_VEL
LIN {X 0,Y 393.266,Z 549.555,A -85,B 0,C 180,E1 10411.558,E2 10411.558} C_VEL
LIN {X 0,Y 402.908,Z 578.911,A -85,B 0,C 180,E1 10413.109,E2 10413.109} C_VEL
LIN {X 0,Y 404.096,Z 592.121,A -85,B 0,C 180,E1 10413.513,E2 10413.513} C_VEL
LIN {X 0,Y 403.962,Z 628.456,A -85,B 0,C 180,E1 10414.589,E2 10414.589} C_VEL
LIN {X 0,Y 403.165,Z 657.002,A -85,B 0,C 180,E1 10416.298,E2 10416.298} C_VEL
LIN {X 0,Y 401.862,Z 681.577,A -85,B 0,C 180,E1 10418.674,E2 10418.674} C_VEL
LIN {X 0,Y 400.342,Z 701.5,A -85,B 0,C 180,E1 10421.603,E2 10421.603} C_VEL
LIN {X 0,Y 398.877,Z 716.307,A -85,B 0,C 180,E1 10424.872,E2 10424.872} C_VEL
LIN {X 0,Y 397.845,Z 726.328,A -85,B 0,C 180,E1 10428.519,E2 10428.519} C_VEL
LIN {X 0,Y 397.216,Z 730.36,A -85,B 0,C 180,E1 10431.264,E2 10431.264} C_VEL
LIN {X 0,Y 396.919,Z 731.593,A -85,B 0,C 180,E1 10433.456,E2 10433.456} C_VEL
LIN {X 0,Y 396.864,Z 730.309,A -85,B 0,C 180,E1 10436.735,E2 10436.735} C_VEL
LIN {X 0,Y 397.017,Z 724.091,A -85,B 0,C 180,E1 10440.549,E2 10440.549} C_VEL
LIN {X 0,Y 397.615,Z 712.324,A -85,B 0,C 180,E1 10444.358,E2 10444.358} C_VEL
LIN {X 0,Y 398.572,Z 695.042,A -85,B 0,C 180,E1 10447.894,E2 10447.894} C_VEL
LIN {X 0,Y 399.944,Z 673.463,A -85,B 0,C 180,E1 10450.879,E2 10450.879} C_VEL
LIN {X 0,Y 401.344,Z 647.096,A -85,B 0,C 180,E1 10453.32,E2 10453.32} C_VEL
LIN {X 0,Y 402.343,Z 617.565,A -85,B 0,C 180,E1 10455.017,E2 10455.017} C_VEL
LIN {X 0,Y 402.404,Z 583.065,A -85,B 0,C 180,E1 10456.005,E2 10456.005} C_VEL
LIN {X 0,Y 393.787,Z 549.53,A -85,B 0,C 180,E1 10457.223,E2 10457.223} C_VEL
LIN {X 0,Y 393.441,Z 549.53,A -85,B 0,C 180,E1 10462.987,E2 10462.987} C_VEL
LIN {X 0,Y 393.189,Z 549.53,A -85,B 0,C 180,E1 10469.935,E2 10469.935} C_VEL
LIN {X 0,Y 392.974,Z 549.53,A -85,B 0,C 180,E1 10476.247,E2 10476.247} C_VEL
LIN {X 0,Y 392.967,Z 549.53,A -85,B 0,C 180,E1 10483.14,E2 10483.14} C_VEL
LIN {X 0,Y 393.056,Z 549.53,A -85,B 0,C 180,E1 10490.169,E2 10490.169} C_VEL
LIN {X 0,Y 393.057,Z 549.545,A -85,B 0,C 180,E1 10492.27,E2 10492.27} C_VEL
LIN {X 0,Y 397.589,Z 559.596,A -85,B 0,C 180,E1 10493.238,E2 10493.238} C_VEL
LIN {X 0,Y 414.306,Z 595.973,A -85,B 0,C 180,E1 10496.556,E2 10496.556} C_VEL
LIN {X 0,Y 419.456,Z 613.739,A -85,B 0,C 180,E1 10498.022,E2 10498.022} C_VEL
LIN {X 0,Y 415.378,Z 649.213,A -85,B 0,C 180,E1 10500.23,E2 10500.23} C_VEL
LIN {X 0,Y 410.341,Z 682.127,A -85,B 0,C 180,E1 10503.222,E2 10503.222} C_VEL
LIN {X 0,Y 405.321,Z 711.763,A -85,B 0,C 180,E1 10506.986,E2 10506.986} C_VEL
LIN {X 0,Y 400.979,Z 736.659,A -85,B 0,C 180,E1 10511.343,E2 10511.343} C_VEL
LIN {X 0,Y 397.885,Z 755.786,A -85,B 0,C 180,E1 10515.952,E2 10515.952} C_VEL
LIN {X 0,Y 395.989,Z 770.843,A -85,B 0,C 180,E1 10521.232,E2 10521.232} C_VEL
LIN {X 0,Y 395.293,Z 778.842,A -85,B 0,C 180,E1 10525.621,E2 10525.621} C_VEL
LIN {X 0,Y 395.095,Z 783.122,A -85,B 0,C 180,E1 10530,E2 10530} C_VEL
LIN {X 0,Y 394.926,Z 783.804,A -85,B 0,C 180,E1 10534.384,E2 10534.384} C_VEL
LIN {X 0,Y 395.169,Z 779.53,A -85,B 0,C 180,E1 10539.896,E2 10539.896} C_VEL
LIN {X 0,Y 396.015,Z 770.601,A -85,B 0,C 180,E1 10544.907,E2 10544.907} C_VEL
LIN {X 0,Y 397.981,Z 756.284,A -85,B 0,C 180,E1 10549.956,E2 10549.956} C_VEL
LIN {X 0,Y 401.27,Z 736.482,A -85,B 0,C 180,E1 10554.777,E2 10554.777} C_VEL
LIN {X 0,Y 405.793,Z 711.875,A -85,B 0,C 180,E1 10559.106,E2 10559.106} C_VEL
LIN {X 0,Y 410.931,Z 683.119,A -85,B 0,C 180,E1 10562.794,E2 10562.794} C_VEL
LIN {X 0,Y 416.063,Z 650.683,A -85,B 0,C 180,E1 10565.796,E2 10565.796} C_VEL
LIN {X 0,Y 420.426,Z 614.931,A -85,B 0,C 180,E1 10568.063,E2 10568.063} C_VEL
LIN {X 0,Y 417.82,Z 602.662,A -85,B 0,C 180,E1 10569.05,E2 10569.05} C_VEL
LIN {X 0,Y 406.002,Z 574.974,A -85,B 0,C 180,E1 10571.644,E2 10571.644} C_VEL
LIN {X 0,Y 393.152,Z 550.67,A -85,B 0,C 180,E1 10574.358,E2 10574.358} C_VEL
LIN {X 0,Y 393.037,Z 549.53,A -85,B 0,C 180,E1 10574.524,E2 10574.524} C_VEL
LIN {X 0,Y 393.194,Z 549.53,A -85,B 0,C 180,E1 10582.11,E2 10582.11} C_VEL
LIN {X 0,Y 393.284,Z 549.53,A -85,B 0,C 180,E1 10587.589,E2 10587.589} C_VEL
LIN {X 0,Y 393.302,Z 549.53,A -85,B 0,C 180,E1 10595.03,E2 10595.03} C_VEL
LIN {X 0,Y 393.477,Z 549.53,A -85,B 0,C 180,E1 10596.553,E2 10596.553} C_VEL
LIN {X 0,Y 401.215,Z 583.173,A -85,B 0,C 180,E1 10597.627,E2 10597.627} C_VEL
LIN {X 0,Y 400.839,Z 633.081,A -85,B 0,C 180,E1 10598.796,E2 10598.796} C_VEL
LIN {X 0,Y 400.171,Z 659.416,A -85,B 0,C 180,E1 10600.239,E2 10600.239} C_VEL
LIN {X 0,Y 399.255,Z 682.838,A -85,B 0,C 180,E1 10602.395,E2 10602.395} C_VEL
LIN {X 0,Y 398.178,Z 702.296,A -85,B 0,C 180,E1 10605.13,E2 10605.13} C_VEL
LIN {X 0,Y 397.393,Z 717.774,A -85,B 0,C 180,E1 10608.495,E2 10608.495} C_VEL
LIN {X 0,Y 396.976,Z 726.594,A -85,B 0,C 180,E1 10611.647,E2 10611.647} C_VEL
LIN {X 0,Y 396.886,Z 729.633,A -85,B 0,C 180,E1 10613.445,E2 10613.445} C_VEL
LIN {X 0,Y 396.951,Z 731.54,A -85,B 0,C 180,E1 10615.635,E2 10615.635} C_VEL
LIN {X 0,Y 397.028,Z 731.54,A -85,B 0,C 180,E1 10617.817,E2 10617.817} C_VEL
LIN {X 0,Y 397.657,Z 726.753,A -85,B 0,C 180,E1 10621.626,E2 10621.626} C_VEL
LIN {X 0,Y 398.685,Z 716.236,A -85,B 0,C 180,E1 10625.153,E2 10625.153} C_VEL
LIN {X 0,Y 399.881,Z 701.315,A -85,B 0,C 180,E1 10628.13,E2 10628.13} C_VEL
LIN {X 0,Y 401.105,Z 681.362,A -85,B 0,C 180,E1 10630.7,E2 10630.7} C_VEL
LIN {X 0,Y 402.028,Z 658.113,A -85,B 0,C 180,E1 10632.6,E2 10632.6} C_VEL
LIN {X 0,Y 402.315,Z 632.261,A -85,B 0,C 180,E1 10633.799,E2 10633.799} C_VEL
LIN {X 0,Y 402.175,Z 578.173,A -85,B 0,C 180,E1 10635.079,E2 10635.079} C_VEL
LIN {X 0,Y 393.752,Z 549.53,A -85,B 0,C 180,E1 10636.414,E2 10636.414} C_VEL
LIN {X 0,Y 393.357,Z 549.53,A -85,B 0,C 180,E1 10642.956,E2 10642.956} C_VEL
LIN {X 0,Y 393.112,Z 549.53,A -85,B 0,C 180,E1 10649.93,E2 10649.93} C_VEL
LIN {X 0,Y 393.045,Z 549.53,A -85,B 0,C 180,E1 10656.26,E2 10656.26} C_VEL
LIN {X 0,Y 393.114,Z 550.335,A -85,B 0,C 180,E1 10661.631,E2 10661.631} C_VEL
LIN {X 0,Y 396.102,Z 555.738,A -85,B 0,C 180,E1 10662.241,E2 10662.241} C_VEL
LIN {X 0,Y 416.97,Z 593.952,A -85,B 0,C 180,E1 10666.258,E2 10666.258} C_VEL
LIN {X 0,Y 427.552,Z 627.373,A -85,B 0,C 180,E1 10668.839,E2 10668.839} C_VEL
LIN {X 0,Y 422.323,Z 670.779,A -85,B 0,C 180,E1 10670.879,E2 10670.879} C_VEL
LIN {X 0,Y 416.493,Z 711.065,A -85,B 0,C 180,E1 10673.658,E2 10673.658} C_VEL
LIN {X 0,Y 410.882,Z 746.083,A -85,B 0,C 180,E1 10676.997,E2 10676.997} C_VEL
LIN {X 0,Y 405.43,Z 776.821,A -85,B 0,C 180,E1 10681.058,E2 10681.058} C_VEL
LIN {X 0,Y 401.587,Z 797.651,A -85,B 0,C 180,E1 10684.7,E2 10684.7} C_VEL
LIN {X 0,Y 395.965,Z 807.523,A -85,B 0,C 180,E1 10686.625,E2 10686.625} C_VEL
LIN {X 0,Y 390.652,Z 816.46,A -85,B 0,C 180,E1 10688.685,E2 10688.685} C_VEL
LIN {X 0,Y 388.163,Z 833.913,A -85,B 0,C 180,E1 10694.207,E2 10694.207} C_VEL
LIN {X 0,Y 387.115,Z 845.965,A -85,B 0,C 180,E1 10699.896,E2 10699.896} C_VEL
LIN {X 0,Y 386.715,Z 852.543,A -85,B 0,C 180,E1 10705.523,E2 10705.523} C_VEL
LIN {X 0,Y 386.83,Z 854.194,A -85,B 0,C 180,E1 10710,E2 10710} C_VEL
LIN {X 0,Y 386.732,Z 852.572,A -85,B 0,C 180,E1 10714.476,E2 10714.476} C_VEL
LIN {X 0,Y 387.048,Z 846.022,A -85,B 0,C 180,E1 10720.105,E2 10720.105} C_VEL
LIN {X 0,Y 388.187,Z 834.016,A -85,B 0,C 180,E1 10725.791,E2 10725.791} C_VEL
LIN {X 0,Y 390.652,Z 816.553,A -85,B 0,C 180,E1 10731.319,E2 10731.319} C_VEL
LIN {X 0,Y 394.812,Z 793.671,A -85,B 0,C 180,E1 10736.457,E2 10736.457} C_VEL
LIN {X 0,Y 400.16,Z 765.188,A -85,B 0,C 180,E1 10741.078,E2 10741.078} C_VEL
LIN {X 0,Y 405.76,Z 733.862,A -85,B 0,C 180,E1 10744.764,E2 10744.764} C_VEL
LIN {X 0,Y 411.701,Z 695.993,A -85,B 0,C 180,E1 10747.983,E2 10747.983} C_VEL
LIN {X 0,Y 417.548,Z 652.739,A -85,B 0,C 180,E1 10750.586,E2 10750.586} C_VEL
LIN {X 0,Y 420.209,Z 626.676,A -85,B 0,C 180,E1 10751.737,E2 10751.737} C_VEL
LIN {X 0,Y 407.566,Z 592.189,A -85,B 0,C 180,E1 10754.552,E2 10754.552} C_VEL
LIN {X 0,Y 387.752,Z 555.369,A -85,B 0,C 180,E1 10758.277,E2 10758.277} C_VEL
LIN {X 0,Y 385.285,Z 550.887,A -85,B 0,C 180,E1 10758.759,E2 10758.759} C_VEL
LIN {X 0,Y 385.174,Z 549.53,A -85,B 0,C 180,E1 10758.992,E2 10758.992} C_VEL
LIN {X 0,Y 385.134,Z 549.53,A -85,B 0,C 180,E1 10765.376,E2 10765.376} C_VEL
LIN {X 0,Y 385.331,Z 549.822,A -85,B 0,C 180,E1 10770.842,E2 10770.842} C_VEL
LIN {X 0,Y 395.159,Z 577.736,A -85,B 0,C 180,E1 10772.509,E2 10772.509} C_VEL
LIN {X 0,Y 397.004,Z 590.667,A -85,B 0,C 180,E1 10772.988,E2 10772.988} C_VEL
LIN {X 0,Y 396.779,Z 629.328,A -85,B 0,C 180,E1 10774.14,E2 10774.14} C_VEL
LIN {X 0,Y 395.908,Z 658.45,A -85,B 0,C 180,E1 10775.903,E2 10775.903} C_VEL
LIN {X 0,Y 394.465,Z 683.696,A -85,B 0,C 180,E1 10778.4,E2 10778.4} C_VEL
LIN {X 0,Y 392.877,Z 703.346,A -85,B 0,C 180,E1 10781.357,E2 10781.357} C_VEL
LIN {X 0,Y 391.293,Z 717.814,A -85,B 0,C 180,E1 10784.626,E2 10784.626} C_VEL
LIN {X 0,Y 390.215,Z 727.746,A -85,B 0,C 180,E1 10788.291,E2 10788.291} C_VEL
LIN {X 0,Y 389.523,Z 731.786,A -85,B 0,C 180,E1 10791.091,E2 10791.091} C_VEL
LIN {X 0,Y 389.164,Z 733.021,A -85,B 0,C 180,E1 10793.325,E2 10793.325} C_VEL
LIN {X 0,Y 389.104,Z 731.717,A -85,B 0,C 180,E1 10796.67,E2 10796.67} C_VEL
LIN {X 0,Y 389.231,Z 725.425,A -85,B 0,C 180,E1 10800.56,E2 10800.56} C_VEL
LIN {X 0,Y 389.845,Z 713.576,A -85,B 0,C 180,E1 10804.445,E2 10804.445} C_VEL
LIN {X 0,Y 390.839,Z 696.185,A -85,B 0,C 180,E1 10808.051,E2 10808.051} C_VEL
LIN {X 0,Y 392.345,Z 673.354,A -85,B 0,C 180,E1 10811.218,E2 10811.218} C_VEL
LIN {X 0,Y 393.78,Z 646.068,A -85,B 0,C 180,E1 10813.722,E2 10813.722} C_VEL
LIN {X 0,Y 394.804,Z 616.38,A -85,B 0,C 180,E1 10815.382,E2 10815.382} C_VEL
LIN {X 0,Y 394.327,Z 582.35,A -85,B 0,C 180,E1 10816.353,E2 10816.353} C_VEL
LIN {X 0,Y 385.871,Z 549.53,A -85,B 0,C 180,E1 10817.467,E2 10817.467} C_VEL
LIN {X 0,Y 385.542,Z 549.53,A -85,B 0,C 180,E1 10823.047,E2 10823.047} C_VEL
LIN {X 0,Y 385.216,Z 549.53,A -85,B 0,C 180,E1 10830.62,E2 10830.62} C_VEL
LIN {X 0,Y 385.078,Z 549.53,A -85,B 0,C 180,E1 10836.008,E2 10836.008} C_VEL
LIN {X 0,Y 384.997,Z 549.53,A -85,B 0,C 180,E1 10841.859,E2 10841.859} C_VEL
LIN {X 0,Y 385.051,Z 549.53,A -85,B 0,C 180,E1 10848.218,E2 10848.218} C_VEL
LIN {X 0,Y 385.114,Z 549.813,A -85,B 0,C 180,E1 10851.219,E2 10851.219} C_VEL
LIN {X 0,Y 405.691,Z 593.188,A -85,B 0,C 180,E1 10855.503,E2 10855.503} C_VEL
LIN {X 0,Y 412.841,Z 615.584,A -85,B 0,C 180,E1 10857.471,E2 10857.471} C_VEL
LIN {X 0,Y 408.497,Z 651.28,A -85,B 0,C 180,E1 10859.758,E2 10859.758} C_VEL
LIN {X 0,Y 403.16,Z 684.407,A -85,B 0,C 180,E1 10862.857,E2 10862.857} C_VEL
LIN {X 0,Y 398.107,Z 712.705,A -85,B 0,C 180,E1 10866.545,E2 10866.545} C_VEL
LIN {X 0,Y 393.52,Z 737.529,A -85,B 0,C 180,E1 10870.975,E2 10870.975} C_VEL
LIN {X 0,Y 390.167,Z 757.025,A -85,B 0,C 180,E1 10875.797,E2 10875.797} C_VEL
LIN {X 0,Y 388.203,Z 771.629,A -85,B 0,C 180,E1 10881.054,E2 10881.054} C_VEL
LIN {X 0,Y 387.377,Z 781.028,A -85,B 0,C 180,E1 10886.65,E2 10886.65} C_VEL
LIN {X 0,Y 387.247,Z 783.845,A -85,B 0,C 180,E1 10890,E2 10890} C_VEL
LIN {X 0,Y 387.051,Z 784.506,A -85,B 0,C 180,E1 10894.473,E2 10894.473} C_VEL
LIN {X 0,Y 387.348,Z 780.172,A -85,B 0,C 180,E1 10900.098,E2 10900.098} C_VEL
LIN {X 0,Y 388.435,Z 769.923,A -85,B 0,C 180,E1 10905.782,E2 10905.782} C_VEL
LIN {X 0,Y 390.608,Z 755.11,A -85,B 0,C 180,E1 10910.863,E2 10910.863} C_VEL
LIN {X 0,Y 394.348,Z 734.665,A -85,B 0,C 180,E1 10915.75,E2 10915.75} C_VEL
LIN {X 0,Y 399.295,Z 709.717,A -85,B 0,C 180,E1 10920.053,E2 10920.053} C_VEL
LIN {X 0,Y 404.893,Z 679.75,A -85,B 0,C 180,E1 10923.816,E2 10923.816} C_VEL
LIN {X 0,Y 410.257,Z 646.431,A -85,B 0,C 180,E1 10926.785,E2 10926.785} C_VEL
LIN {X 0,Y 413.706,Z 613.078,A -85,B 0,C 180,E1 10928.916,E2 10928.916} C_VEL
LIN {X 0,Y 404.992,Z 588.673,A -85,B 0,C 180,E1 10931.211,E2 10931.211} C_VEL
LIN {X 0,Y 387.437,Z 555.112,A -85,B 0,C 180,E1 10935.012,E2 10935.012} C_VEL
LIN {X 0,Y 385.092,Z 549.53,A -85,B 0,C 180,E1 10935.732,E2 10935.732} C_VEL
LIN {X 0,Y 385.239,Z 549.53,A -85,B 0,C 180,E1 10941.583,E2 10941.583} C_VEL
LIN {X 0,Y 385.27,Z 549.53,A -85,B 0,C 180,E1 10946.74,E2 10946.74} C_VEL
LIN {X 0,Y 385.299,Z 549.53,A -85,B 0,C 180,E1 10951.961,E2 10951.961} C_VEL
LIN {X 0,Y 385.569,Z 550.308,A -85,B 0,C 180,E1 10956.258,E2 10956.258} C_VEL
LIN {X 0,Y 393.627,Z 585.675,A -85,B 0,C 180,E1 10957.379,E2 10957.379} C_VEL
LIN {X 0,Y 393.177,Z 633.839,A -85,B 0,C 180,E1 10958.534,E2 10958.534} C_VEL
LIN {X 0,Y 392.5,Z 660.043,A -85,B 0,C 180,E1 10959.981,E2 10959.981} C_VEL
LIN {X 0,Y 391.549,Z 683.728,A -85,B 0,C 180,E1 10962.182,E2 10962.182} C_VEL
LIN {X 0,Y 390.348,Z 704.306,A -85,B 0,C 180,E1 10965.143,E2 10965.143} C_VEL
LIN {X 0,Y 389.636,Z 718.442,A -85,B 0,C 180,E1 10968.263,E2 10968.263} C_VEL
LIN {X 0,Y 389.213,Z 727.583,A -85,B 0,C 180,E1 10971.479,E2 10971.479} C_VEL
LIN {X 0,Y 389.114,Z 732.046,A -85,B 0,C 180,E1 10974.431,E2 10974.431} C_VEL
LIN {X 0,Y 389.261,Z 732.969,A -85,B 0,C 180,E1 10977.773,E2 10977.773} C_VEL
LIN {X 0,Y 389.933,Z 728.406,A -85,B 0,C 180,E1 10981.658,E2 10981.658} C_VEL
LIN {X 0,Y 391.016,Z 718.112,A -85,B 0,C 180,E1 10985.254,E2 10985.254} C_VEL
LIN {X 0,Y 392.307,Z 703.414,A -85,B 0,C 180,E1 10988.288,E2 10988.288} C_VEL
LIN {X 0,Y 393.614,Z 683.862,A -85,B 0,C 180,E1 10990.906,E2 10990.906} C_VEL
LIN {X 0,Y 394.613,Z 659.996,A -85,B 0,C 180,E1 10992.922,E2 10992.922} C_VEL
LIN {X 0,Y 394.963,Z 633.084,A -85,B 0,C 180,E1 10994.188,E2 10994.188} C_VEL
LIN {X 0,Y 394.824,Z 579.258,A -85,B 0,C 180,E1 10995.513,E2 10995.513} C_VEL
LIN {X 0,Y 385.772,Z 549.53,A -85,B 0,C 180,E1 10996.961,E2 10996.961} C_VEL
LIN {X 0,Y 385.457,Z 549.53,A -85,B 0,C 180,E1 11003.042,E2 11003.042} C_VEL
LIN {X 0,Y 385.162,Z 549.53,A -85,B 0,C 180,E1 11010.613,E2 11010.613} C_VEL
LIN {X 0,Y 385.184,Z 549.53,A -85,B 0,C 180,E1 11018.407,E2 11018.407} C_VEL
LIN {X 0,Y 385.192,Z 549.53,A -85,B 0,C 180,E1 11020.322,E2 11020.322} C_VEL
LIN {X 0,Y 387.689,Z 555.313,A -85,B 0,C 180,E1 11020.927,E2 11020.927} C_VEL
LIN {X 0,Y 407.303,Z 589.76,A -85,B 0,C 180,E1 11024.908,E2 11024.908} C_VEL
LIN {X 0,Y 413.912,Z 606.302,A -85,B 0,C 180,E1 11026.391,E2 11026.391} C_VEL
LIN {X 0,Y 420.906,Z 630.792,A -85,B 0,C 180,E1 11028.326,E2 11028.326} C_VEL
LIN {X 0,Y 415.382,Z 673.63,A -85,B 0,C 180,E1 11030.435,E2 11030.435} C_VEL
LIN {X 0,Y 409.114,Z 714.903,A -85,B 0,C 180,E1 11033.406,E2 11033.406} C_VEL
LIN {X 0,Y 403.238,Z 749.101,A -85,B 0,C 180,E1 11036.824,E2 11036.824} C_VEL
LIN {X 0,Y 397.757,Z 778.358,A -85,B 0,C 180,E1 11040.861,E2 11040.861} C_VEL
LIN {X 0,Y 392.907,Z 803.742,A -85,B 0,C 180,E1 11045.612,E2 11045.612} C_VEL
LIN {X 0,Y 390.652,Z 816.46,A -85,B 0,C 180,E1 11048.685,E2 11048.685} C_VEL
LIN {X 0,Y 387.302,Z 822.554,A -85,B 0,C 180,E1 11050.33,E2 11050.33} C_VEL
LIN {X 0,Y 380.784,Z 830.575,A -85,B 0,C 180,E1 11052.861,E2 11052.861} C_VEL
LIN {X 0,Y 380.576,Z 831.415,A -85,B 0,C 180,E1 11053.165,E2 11053.165} C_VEL
LIN {X 0,Y 379.382,Z 843.345,A -85,B 0,C 180,E1 11058.527,E2 11058.527} C_VEL
LIN {X 0,Y 378.974,Z 849.843,A -85,B 0,C 180,E1 11063.138,E2 11063.138} C_VEL
LIN {X 0,Y 378.885,Z 853.057,A -85,B 0,C 180,E1 11067.717,E2 11067.717} C_VEL
LIN {X 0,Y 378.931,Z 853.079,A -85,B 0,C 180,E1 11072.282,E2 11072.282} C_VEL
LIN {X 0,Y 379.015,Z 848.593,A -85,B 0,C 180,E1 11078.011,E2 11078.011} C_VEL
LIN {X 0,Y 379.741,Z 838.862,A -85,B 0,C 180,E1 11083.795,E2 11083.795} C_VEL
LIN {X 0,Y 381.501,Z 825.102,A -85,B 0,C 180,E1 11089.048,E2 11089.048} C_VEL
LIN {X 0,Y 385.138,Z 804.253,A -85,B 0,C 180,E1 11094.604,E2 11094.604} C_VEL
LIN {X 0,Y 390.182,Z 778.706,A -85,B 0,C 180,E1 11099.489,E2 11099.489} C_VEL
LIN {X 0,Y 395.965,Z 749.039,A -85,B 0,C 180,E1 11103.63,E2 11103.63} C_VEL
LIN {X 0,Y 401.906,Z 715.061,A -85,B 0,C 180,E1 11107.042,E2 11107.042} C_VEL
LIN {X 0,Y 408.105,Z 674.406,A -85,B 0,C 180,E1 11110,E2 11110} C_VEL
LIN {X 0,Y 413.76,Z 631.074,A -85,B 0,C 180,E1 11112.161,E2 11112.161} C_VEL
LIN {X 0,Y 402.497,Z 597.72,A -85,B 0,C 180,E1 11114.924,E2 11114.924} C_VEL
LIN {X 0,Y 383.388,Z 561.276,A -85,B 0,C 180,E1 11118.74,E2 11118.74} C_VEL
LIN {X 0,Y 377.314,Z 550.533,A -85,B 0,C 180,E1 11119.972,E2 11119.972} C_VEL
LIN {X 0,Y 377.235,Z 549.53,A -85,B 0,C 180,E1 11120.212,E2 11120.212} C_VEL
LIN {X 0,Y 377.203,Z 549.53,A -85,B 0,C 180,E1 11127.161,E2 11127.161} C_VEL
LIN {X 0,Y 377.368,Z 549.901,A -85,B 0,C 180,E1 11130.033,E2 11130.033} C_VEL
LIN {X 0,Y 387.989,Z 578.459,A -85,B 0,C 180,E1 11131.952,E2 11131.952} C_VEL
LIN {X 0,Y 389.98,Z 590.829,A -85,B 0,C 180,E1 11132.461,E2 11132.461} C_VEL
LIN {X 0,Y 389.616,Z 631.484,A -85,B 0,C 180,E1 11133.722,E2 11133.722} C_VEL
LIN {X 0,Y 388.713,Z 660.308,A -85,B 0,C 180,E1 11135.514,E2 11135.514} C_VEL
LIN {X 0,Y 387.205,Z 684.815,A -85,B 0,C 180,E1 11137.975,E2 11137.975} C_VEL
LIN {X 0,Y 385.472,Z 704.547,A -85,B 0,C 180,E1 11140.975,E2 11140.975} C_VEL
LIN {X 0,Y 383.767,Z 719.328,A -85,B 0,C 180,E1 11144.353,E2 11144.353} C_VEL
LIN {X 0,Y 382.583,Z 729.167,A -85,B 0,C 180,E1 11148.054,E2 11148.054} C_VEL
LIN {X 0,Y 381.774,Z 733.476,A -85,B 0,C 180,E1 11151.212,E2 11151.212} C_VEL
LIN {X 0,Y 381.38,Z 733.992,A -85,B 0,C 180,E1 11155.466,E2 11155.466} C_VEL
LIN {X 0,Y 381.369,Z 729.138,A -85,B 0,C 180,E1 11159.438,E2 11159.438} C_VEL
LIN {X 0,Y 381.735,Z 718.848,A -85,B 0,C 180,E1 11163.405,E2 11163.405} C_VEL
LIN {X 0,Y 382.695,Z 703.474,A -85,B 0,C 180,E1 11167.083,E2 11167.083} C_VEL
LIN {X 0,Y 384.11,Z 682.153,A -85,B 0,C 180,E1 11170.473,E2 11170.473} C_VEL
LIN {X 0,Y 385.621,Z 657.151,A -85,B 0,C 180,E1 11173.153,E2 11173.153} C_VEL
LIN {X 0,Y 386.853,Z 628.667,A -85,B 0,C 180,E1 11175.127,E2 11175.127} C_VEL
LIN {X 0,Y 387.508,Z 596.489,A -85,B 0,C 180,E1 11176.319,E2 11176.319} C_VEL
LIN {X 0,Y 386.385,Z 582.168,A -85,B 0,C 180,E1 11176.695,E2 11176.695} C_VEL
LIN {X 0,Y 377.887,Z 549.53,A -85,B 0,C 180,E1 11177.898,E2 11177.898} C_VEL
LIN {X 0,Y 377.564,Z 549.53,A -85,B 0,C 180,E1 11183.564,E2 11183.564} C_VEL
LIN {X 0,Y 377.352,Z 549.53,A -85,B 0,C 180,E1 11188.683,E2 11188.683} C_VEL
LIN {X 0,Y 377.148,Z 549.53,A -85,B 0,C 180,E1 11194.073,E2 11194.073} C_VEL
LIN {X 0,Y 377.017,Z 549.53,A -85,B 0,C 180,E1 11200.487,E2 11200.487} C_VEL
LIN {X 0,Y 377.035,Z 549.53,A -85,B 0,C 180,E1 11207.12,E2 11207.12} C_VEL
LIN {X 0,Y 377.117,Z 550.213,A -85,B 0,C 180,E1 11210.095,E2 11210.095} C_VEL
LIN {X 0,Y 397.369,Z 591.267,A -85,B 0,C 180,E1 11214.482,E2 11214.482} C_VEL
LIN {X 0,Y 406.253,Z 617.058,A -85,B 0,C 180,E1 11216.878,E2 11216.878} C_VEL
LIN {X 0,Y 401.871,Z 651.863,A -85,B 0,C 180,E1 11219.147,E2 11219.147} C_VEL
LIN {X 0,Y 396.448,Z 684.209,A -85,B 0,C 180,E1 11222.204,E2 11222.204} C_VEL
LIN {X 0,Y 390.896,Z 713.661,A -85,B 0,C 180,E1 11226.085,E2 11226.085} C_VEL
LIN {X 0,Y 386.062,Z 738.412,A -85,B 0,C 180,E1 11230.593,E2 11230.593} C_VEL
LIN {X 0,Y 382.448,Z 758.348,A -85,B 0,C 180,E1 11235.661,E2 11235.661} C_VEL
LIN {X 0,Y 380.422,Z 772.417,A -85,B 0,C 180,E1 11240.87,E2 11240.87} C_VEL
LIN {X 0,Y 379.522,Z 781.777,A -85,B 0,C 180,E1 11246.581,E2 11246.581} C_VEL
LIN {X 0,Y 379.397,Z 784.569,A -85,B 0,C 180,E1 11250,E2 11250} C_VEL
LIN {X 0,Y 379.127,Z 784.79,A -85,B 0,C 180,E1 11255.64,E2 11255.64} C_VEL
LIN {X 0,Y 379.704,Z 779.292,A -85,B 0,C 180,E1 11261.463,E2 11261.463} C_VEL
LIN {X 0,Y 380.919,Z 769.131,A -85,B 0,C 180,E1 11266.684,E2 11266.684} C_VEL
LIN {X 0,Y 383.655,Z 752.717,A -85,B 0,C 180,E1 11272.125,E2 11272.125} C_VEL
LIN {X 0,Y 388.062,Z 730.862,A -85,B 0,C 180,E1 11277.117,E2 11277.117} C_VEL
LIN {X 0,Y 393.627,Z 704.255,A -85,B 0,C 180,E1 11281.493,E2 11281.493} C_VEL
LIN {X 0,Y 399.366,Z 674.043,A -85,B 0,C 180,E1 11285.081,E2 11285.081} C_VEL
LIN {X 0,Y 404.924,Z 640.179,A -85,B 0,C 180,E1 11287.922,E2 11287.922} C_VEL
LIN {X 0,Y 407.277,Z 615.723,A -85,B 0,C 180,E1 11289.482,E2 11289.482} C_VEL
LIN {X 0,Y 398.817,Z 591.837,A -85,B 0,C 180,E1 11291.84,E2 11291.84} C_VEL
LIN {X 0,Y 382.377,Z 560.344,A -85,B 0,C 180,E1 11295.549,E2 11295.549} C_VEL
LIN {X 0,Y 377.262,Z 550.322,A -85,B 0,C 180,E1 11296.842,E2 11296.842} C_VEL
LIN {X 0,Y 377.304,Z 549.53,A -85,B 0,C 180,E1 11303.129,E2 11303.129} C_VEL
LIN {X 0,Y 377.318,Z 549.53,A -85,B 0,C 180,E1 11308.667,E2 11308.667} C_VEL
LIN {X 0,Y 377.6,Z 549.53,A -85,B 0,C 180,E1 11315.873,E2 11315.873} C_VEL
LIN {X 0,Y 386,Z 584.552,A -85,B 0,C 180,E1 11317.054,E2 11317.054} C_VEL
LIN {X 0,Y 385.489,Z 636.134,A -85,B 0,C 180,E1 11318.336,E2 11318.336} C_VEL
LIN {X 0,Y 384.741,Z 663.518,A -85,B 0,C 180,E1 11319.941,E2 11319.941} C_VEL
LIN {X 0,Y 383.752,Z 686.952,A -85,B 0,C 180,E1 11322.251,E2 11322.251} C_VEL
LIN {X 0,Y 382.54,Z 706.114,A -85,B 0,C 180,E1 11325.125,E2 11325.125} C_VEL
LIN {X 0,Y 381.789,Z 721.094,A -85,B 0,C 180,E1 11328.597,E2 11328.597} C_VEL
LIN {X 0,Y 381.334,Z 730.501,A -85,B 0,C 180,E1 11332.337,E2 11332.337} C_VEL
LIN {X 0,Y 381.403,Z 734.105,A -85,B 0,C 180,E1 11335.456,E2 11335.456} C_VEL
LIN {X 0,Y 381.494,Z 734.384,A -85,B 0,C 180,E1 11337.728,E2 11337.728} C_VEL
LIN {X 0,Y 382.223,Z 730.06,A -85,B 0,C 180,E1 11341.692,E2 11341.692} C_VEL
LIN {X 0,Y 383.354,Z 720.005,A -85,B 0,C 180,E1 11345.359,E2 11345.359} C_VEL
LIN {X 0,Y 384.746,Z 705.615,A -85,B 0,C 180,E1 11348.453,E2 11348.453} C_VEL
LIN {X 0,Y 386.129,Z 686.389,A -85,B 0,C 180,E1 11351.12,E2 11351.12} C_VEL
LIN {X 0,Y 387.246,Z 661.998,A -85,B 0,C 180,E1 11353.257,E2 11353.257} C_VEL
LIN {X 0,Y 387.671,Z 635.105,A -85,B 0,C 180,E1 11354.567,E2 11354.567} C_VEL
LIN {X 0,Y 387.567,Z 580.452,A -85,B 0,C 180,E1 11355.975,E2 11355.975} C_VEL
LIN {X 0,Y 378.403,Z 552.524,A -85,B 0,C 180,E1 11357.444,E2 11357.444} C_VEL
LIN {X 0,Y 377.788,Z 549.53,A -85,B 0,C 180,E1 11357.621,E2 11357.621} C_VEL
LIN {X 0,Y 377.492,Z 549.53,A -85,B 0,C 180,E1 11363.557,E2 11363.557} C_VEL
LIN {X 0,Y 377.246,Z 549.53,A -85,B 0,C 180,E1 11368.68,E2 11368.68} C_VEL
LIN {X 0,Y 377.155,Z 549.53,A -85,B 0,C 180,E1 11374.06,E2 11374.06} C_VEL
LIN {X 0,Y 377.3,Z 549.53,A -85,B 0,C 180,E1 11378.972,E2 11378.972} C_VEL
LIN {X 0,Y 379.595,Z 555.101,A -85,B 0,C 180,E1 11379.578,E2 11379.578} C_VEL
LIN {X 0,Y 398.568,Z 587.69,A -85,B 0,C 180,E1 11383.672,E2 11383.672} C_VEL
LIN {X 0,Y 407.419,Z 607.767,A -85,B 0,C 180,E1 11385.673,E2 11385.673} C_VEL
LIN {X 0,Y 414.435,Z 632.843,A -85,B 0,C 180,E1 11387.737,E2 11387.737} C_VEL
LIN {X 0,Y 408.604,Z 675.579,A -85,B 0,C 180,E1 11389.92,E2 11389.92} C_VEL
LIN {X 0,Y 402.032,Z 716.571,A -85,B 0,C 180,E1 11392.964,E2 11392.964} C_VEL
LIN {X 0,Y 396.021,Z 749.812,A -85,B 0,C 180,E1 11396.377,E2 11396.377} C_VEL
LIN {X 0,Y 390.274,Z 778.99,A -85,B 0,C 180,E1 11400.512,E2 11400.512} C_VEL
LIN {X 0,Y 385.163,Z 804.276,A -85,B 0,C 180,E1 11405.397,E2 11405.397} C_VEL
LIN {X 0,Y 381.503,Z 825.01,A -85,B 0,C 180,E1 11410.952,E2 11410.952} C_VEL
LIN {X 0,Y 380.576,Z 831.415,A -85,B 0,C 180,E1 11413.165,E2 11413.165} C_VEL
LIN {X 0,Y 375.941,Z 837.367,A -85,B 0,C 180,E1 11415.562,E2 11415.562} C_VEL
LIN {X 0,Y 371.538,Z 842.278,A -85,B 0,C 180,E1 11418.068,E2 11418.068} C_VEL
LIN {X 0,Y 371.088,Z 849.153,A -85,B 0,C 180,E1 11422.992,E2 11422.992} C_VEL
LIN {X 0,Y 371.004,Z 852.35,A -85,B 0,C 180,E1 11427.668,E2 11427.668} C_VEL
LIN {X 0,Y 371.049,Z 852.374,A -85,B 0,C 180,E1 11432.331,E2 11432.331} C_VEL
LIN {X 0,Y 371.141,Z 847.914,A -85,B 0,C 180,E1 11438.182,E2 11438.182} C_VEL
LIN {X 0,Y 371.927,Z 838.162,A -85,B 0,C 180,E1 11444.091,E2 11444.091} C_VEL
LIN {X 0,Y 373.801,Z 824.332,A -85,B 0,C 180,E1 11449.456,E2 11449.456} C_VEL
LIN {X 0,Y 377.398,Z 804.639,A -85,B 0,C 180,E1 11454.827,E2 11454.827} C_VEL
LIN {X 0,Y 382.663,Z 779.253,A -85,B 0,C 180,E1 11459.833,E2 11459.833} C_VEL
LIN {X 0,Y 388.627,Z 750.012,A -85,B 0,C 180,E1 11464.022,E2 11464.022} C_VEL
LIN {X 0,Y 394.727,Z 717.024,A -85,B 0,C 180,E1 11467.447,E2 11467.447} C_VEL
LIN {X 0,Y 401.154,Z 676.743,A -85,B 0,C 180,E1 11470.475,E2 11470.475} C_VEL
LIN {X 0,Y 406.682,Z 631.367,A -85,B 0,C 180,E1 11472.873,E2 11472.873} C_VEL
LIN {X 0,Y 396.373,Z 601.007,A -85,B 0,C 180,E1 11475.52,E2 11475.52} C_VEL
LIN {X 0,Y 378.453,Z 566.49,A -85,B 0,C 180,E1 11479.292,E2 11479.292} C_VEL
LIN {X 0,Y 369.305,Z 550.674,A -85,B 0,C 180,E1 11481.258,E2 11481.258} C_VEL
LIN {X 0,Y 369.229,Z 549.53,A -85,B 0,C 180,E1 11481.321,E2 11481.321} C_VEL
LIN {X 0,Y 369.346,Z 549.628,A -85,B 0,C 180,E1 11489.101,E2 11489.101} C_VEL
LIN {X 0,Y 380.76,Z 578.838,A -85,B 0,C 180,E1 11491.327,E2 11491.327} C_VEL
LIN {X 0,Y 383.046,Z 592.828,A -85,B 0,C 180,E1 11491.948,E2 11491.948} C_VEL
LIN {X 0,Y 382.559,Z 634.194,A -85,B 0,C 180,E1 11493.298,E2 11493.298} C_VEL
LIN {X 0,Y 381.553,Z 662.141,A -85,B 0,C 180,E1 11495.099,E2 11495.099} C_VEL
LIN {X 0,Y 379.865,Z 687.192,A -85,B 0,C 180,E1 11497.68,E2 11497.68} C_VEL
LIN {X 0,Y 377.921,Z 707.74,A -85,B 0,C 180,E1 11500.938,E2 11500.938} C_VEL
LIN {X 0,Y 376.109,Z 721.873,A -85,B 0,C 180,E1 11504.369,E2 11504.369} C_VEL
LIN {X 0,Y 374.779,Z 731.659,A -85,B 0,C 180,E1 11508.391,E2 11508.391} C_VEL
LIN {X 0,Y 374.156,Z 734.698,A -85,B 0,C 180,E1 11510.721,E2 11510.721} C_VEL
LIN {X 0,Y 373.693,Z 735.91,A -85,B 0,C 180,E1 11513.047,E2 11513.047} C_VEL
LIN {X 0,Y 373.536,Z 734.539,A -85,B 0,C 180,E1 11516.531,E2 11516.531} C_VEL
LIN {X 0,Y 373.649,Z 728.089,A -85,B 0,C 180,E1 11520.584,E2 11520.584} C_VEL
LIN {X 0,Y 374.307,Z 716.014,A -85,B 0,C 180,E1 11524.63,E2 11524.63} C_VEL
LIN {X 0,Y 375.348,Z 698.308,A -85,B 0,C 180,E1 11528.385,E2 11528.385} C_VEL
LIN {X 0,Y 376.876,Z 676.156,A -85,B 0,C 180,E1 11531.554,E2 11531.554} C_VEL
LIN {X 0,Y 378.434,Z 649.092,A -85,B 0,C 180,E1 11534.142,E2 11534.142} C_VEL
LIN {X 0,Y 379.514,Z 619.879,A -85,B 0,C 180,E1 11535.87,E2 11535.87} C_VEL
LIN {X 0,Y 379.164,Z 585.019,A -85,B 0,C 180,E1 11536.937,E2 11536.937} C_VEL
LIN {X 0,Y 369.938,Z 549.53,A -85,B 0,C 180,E1 11538.251,E2 11538.251} C_VEL
LIN {X 0,Y 369.532,Z 549.53,A -85,B 0,C 180,E1 11546.041,E2 11546.041} C_VEL
LIN {X 0,Y 369.249,Z 549.53,A -85,B 0,C 180,E1 11552.098,E2 11552.098} C_VEL
LIN {X 0,Y 369.042,Z 549.53,A -85,B 0,C 180,E1 11559.014,E2 11559.014} C_VEL
LIN {X 0,Y 369.099,Z 549.53,A -85,B 0,C 180,E1 11565.965,E2 11565.965} C_VEL
LIN {X 0,Y 369.096,Z 549.53,A -85,B 0,C 180,E1 11568.842,E2 11568.842} C_VEL
LIN {X 0,Y 371.417,Z 555.039,A -85,B 0,C 180,E1 11569.459,E2 11569.459} C_VEL
LIN {X 0,Y 388.791,Z 589.149,A -85,B 0,C 180,E1 11573.361,E2 11573.361} C_VEL
LIN {X 0,Y 398.983,Z 616.974,A -85,B 0,C 180,E1 11576.079,E2 11576.079} C_VEL
LIN {X 0,Y 399.013,Z 625.664,A -85,B 0,C 180,E1 11576.675,E2 11576.675} C_VEL
LIN {X 0,Y 393.959,Z 660.558,A -85,B 0,C 180,E1 11579.198,E2 11579.198} C_VEL
LIN {X 0,Y 388.121,Z 692.559,A -85,B 0,C 180,E1 11582.527,E2 11582.527} C_VEL
LIN {X 0,Y 382.662,Z 719.87,A -85,B 0,C 180,E1 11586.465,E2 11586.465} C_VEL
LIN {X 0,Y 377.849,Z 743.215,A -85,B 0,C 180,E1 11591.083,E2 11591.083} C_VEL
LIN {X 0,Y 374.464,Z 761.196,A -85,B 0,C 180,E1 11596.007,E2 11596.007} C_VEL
LIN {X 0,Y 372.49,Z 774.465,A -85,B 0,C 180,E1 11601.261,E2 11601.261} C_VEL
LIN {X 0,Y 371.692,Z 782.523,A -85,B 0,C 180,E1 11606.509,E2 11606.509} C_VEL
LIN {X 0,Y 371.544,Z 785.292,A -85,B 0,C 180,E1 11610,E2 11610} C_VEL
LIN {X 0,Y 371.334,Z 785.909,A -85,B 0,C 180,E1 11614.663,E2 11614.663} C_VEL
LIN {X 0,Y 371.718,Z 781.472,A -85,B 0,C 180,E1 11620.528,E2 11620.528} C_VEL
LIN {X 0,Y 372.835,Z 772.424,A -85,B 0,C 180,E1 11625.857,E2 11625.857} C_VEL
LIN {X 0,Y 375.304,Z 757.992,A -85,B 0,C 180,E1 11631.218,E2 11631.218} C_VEL
LIN {X 0,Y 379.461,Z 737.605,A -85,B 0,C 180,E1 11636.398,E2 11636.398} C_VEL
LIN {X 0,Y 385.068,Z 712.529,A -85,B 0,C 180,E1 11640.958,E2 11640.958} C_VEL
LIN {X 0,Y 390.88,Z 684.644,A -85,B 0,C 180,E1 11644.653,E2 11644.653} C_VEL
LIN {X 0,Y 396.75,Z 652.283,A -85,B 0,C 180,E1 11647.751,E2 11647.751} C_VEL
LIN {X 0,Y 401.075,Z 619.046,A -85,B 0,C 180,E1 11649.996,E2 11649.996} C_VEL
LIN {X 0,Y 392.708,Z 594.877,A -85,B 0,C 180,E1 11652.49,E2 11652.49} C_VEL
LIN {X 0,Y 376.58,Z 564.014,A -85,B 0,C 180,E1 11656.295,E2 11656.295} C_VEL
LIN {X 0,Y 369.234,Z 549.989,A -85,B 0,C 180,E1 11658.251,E2 11658.251} C_VEL
LIN {X 0,Y 369.329,Z 549.53,A -85,B 0,C 180,E1 11665.102,E2 11665.102} C_VEL
LIN {X 0,Y 369.376,Z 549.53,A -85,B 0,C 180,E1 11670.637,E2 11670.637} C_VEL
LIN {X 0,Y 369.66,Z 549.53,A -85,B 0,C 180,E1 11675.502,E2 11675.502} C_VEL
LIN {X 0,Y 378.388,Z 588.024,A -85,B 0,C 180,E1 11676.82,E2 11676.82} C_VEL
LIN {X 0,Y 377.856,Z 636.828,A -85,B 0,C 180,E1 11678.064,E2 11678.064} C_VEL
LIN {X 0,Y 377.093,Z 663.764,A -85,B 0,C 180,E1 11679.648,E2 11679.648} C_VEL
LIN {X 0,Y 376.039,Z 687.773,A -85,B 0,C 180,E1 11682.026,E2 11682.026} C_VEL
LIN {X 0,Y 374.707,Z 708.185,A -85,B 0,C 180,E1 11685.158,E2 11685.158} C_VEL
LIN {X 0,Y 374.034,Z 721.775,A -85,B 0,C 180,E1 11688.357,E2 11688.357} C_VEL
LIN {X 0,Y 373.56,Z 731.811,A -85,B 0,C 180,E1 11692.324,E2 11692.324} C_VEL
LIN {X 0,Y 373.633,Z 735.361,A -85,B 0,C 180,E1 11695.362,E2 11695.362} C_VEL
LIN {X 0,Y 373.718,Z 735.794,A -85,B 0,C 180,E1 11697.681,E2 11697.681} C_VEL
LIN {X 0,Y 374.499,Z 731.731,A -85,B 0,C 180,E1 11701.727,E2 11701.727} C_VEL
LIN {X 0,Y 375.704,Z 721.951,A -85,B 0,C 180,E1 11705.469,E2 11705.469} C_VEL
LIN {X 0,Y 377.192,Z 707.815,A -85,B 0,C 180,E1 11708.623,E2 11708.623} C_VEL
LIN {X 0,Y 378.753,Z 687.766,A -85,B 0,C 180,E1 11711.485,E2 11711.485} C_VEL
LIN {X 0,Y 379.928,Z 663.842,A -85,B 0,C 180,E1 11713.622,E2 11713.622} C_VEL
LIN {X 0,Y 380.397,Z 636.487,A -85,B 0,C 180,E1 11714.991,E2 11714.991} C_VEL
LIN {X 0,Y 380.554,Z 582.483,A -85,B 0,C 180,E1 11716.421,E2 11716.421} C_VEL
LIN {X 0,Y 371.466,Z 554.538,A -85,B 0,C 180,E1 11717.981,E2 11717.981} C_VEL
LIN {X 0,Y 369.861,Z 549.53,A -85,B 0,C 180,E1 11718.439,E2 11718.439} C_VEL
LIN {X 0,Y 369.452,Z 549.53,A -85,B 0,C 180,E1 11726.014,E2 11726.014} C_VEL
LIN {X 0,Y 369.219,Z 549.53,A -85,B 0,C 180,E1 11732.088,E2 11732.088} C_VEL
LIN {X 0,Y 369.294,Z 549.53,A -85,B 0,C 180,E1 11737.531,E2 11737.531} C_VEL
LIN {X 0,Y 371.733,Z 555.163,A -85,B 0,C 180,E1 11738.183,E2 11738.183} C_VEL
LIN {X 0,Y 391.219,Z 588.117,A -85,B 0,C 180,E1 11742.656,E2 11742.656} C_VEL
LIN {X 0,Y 401.569,Z 611.356,A -85,B 0,C 180,E1 11745.123,E2 11745.123} C_VEL
LIN {X 0,Y 407.975,Z 634.715,A -85,B 0,C 180,E1 11747.13,E2 11747.13} C_VEL
LIN {X 0,Y 401.804,Z 677.508,A -85,B 0,C 180,E1 11749.395,E2 11749.395} C_VEL
LIN {X 0,Y 395.09,Z 717.6,A -85,B 0,C 180,E1 11752.453,E2 11752.453} C_VEL
LIN {X 0,Y 388.727,Z 751.067,A -85,B 0,C 180,E1 11755.984,E2 11755.984} C_VEL
LIN {X 0,Y 382.622,Z 780.417,A -85,B 0,C 180,E1 11760.291,E2 11760.291} C_VEL
LIN {X 0,Y 377.211,Z 806.082,A -85,B 0,C 180,E1 11765.474,E2 11765.474} C_VEL
LIN {X 0,Y 373.494,Z 826.079,A -85,B 0,C 180,E1 11771.14,E2 11771.14} C_VEL
LIN {X 0,Y 371.698,Z 840.257,A -85,B 0,C 180,E1 11776.973,E2 11776.973} C_VEL
LIN {X 0,Y 371.538,Z 842.278,A -85,B 0,C 180,E1 11778.068,E2 11778.068} C_VEL
LIN {X 0,Y 368.824,Z 845.342,A -85,B 0,C 180,E1 11779.998,E2 11779.998} C_VEL
LIN {X 0,Y 363.143,Z 848.838,A -85,B 0,C 180,E1 11783.296,E2 11783.296} C_VEL
LIN {X 0,Y 363.124,Z 851.644,A -85,B 0,C 180,E1 11787.618,E2 11787.618} C_VEL
LIN {X 0,Y 363.168,Z 851.666,A -85,B 0,C 180,E1 11792.381,E2 11792.381} C_VEL
LIN {X 0,Y 363.255,Z 847.207,A -85,B 0,C 180,E1 11798.361,E2 11798.361} C_VEL
LIN {X 0,Y 364.103,Z 837.421,A -85,B 0,C 180,E1 11804.4,E2 11804.4} C_VEL
LIN {X 0,Y 366.118,Z 823.522,A -85,B 0,C 180,E1 11809.881,E2 11809.881} C_VEL
LIN {X 0,Y 369.901,Z 803.796,A -85,B 0,C 180,E1 11815.347,E2 11815.347} C_VEL
LIN {X 0,Y 375.544,Z 778.174,A -85,B 0,C 180,E1 11820.458,E2 11820.458} C_VEL
LIN {X 0,Y 381.897,Z 748.098,A -85,B 0,C 180,E1 11824.787,E2 11824.787} C_VEL
LIN {X 0,Y 388.217,Z 715.04,A -85,B 0,C 180,E1 11828.214,E2 11828.214} C_VEL
LIN {X 0,Y 395.029,Z 673.923,A -85,B 0,C 180,E1 11831.283,E2 11831.283} C_VEL
LIN {X 0,Y 400.029,Z 633.658,A -85,B 0,C 180,E1 11833.464,E2 11833.464} C_VEL
LIN {X 0,Y 390.862,Z 605.636,A -85,B 0,C 180,E1 11835.985,E2 11835.985} C_VEL
LIN {X 0,Y 373.514,Z 571.563,A -85,B 0,C 180,E1 11839.85,E2 11839.85} C_VEL
LIN {X 0,Y 361.357,Z 550.675,A -85,B 0,C 180,E1 11842.626,E2 11842.626} C_VEL
LIN {X 0,Y 361.247,Z 549.53,A -85,B 0,C 180,E1 11842.815,E2 11842.815} C_VEL
LIN {X 0,Y 361.409,Z 550.176,A -85,B 0,C 180,E1 11848.084,E2 11848.084} C_VEL
LIN {X 0,Y 372.846,Z 576.946,A -85,B 0,C 180,E1 11850.491,E2 11850.491} C_VEL
LIN {X 0,Y 376.261,Z 592.008,A -85,B 0,C 180,E1 11851.317,E2 11851.317} C_VEL
LIN {X 0,Y 375.593,Z 634.635,A -85,B 0,C 180,E1 11852.729,E2 11852.729} C_VEL
LIN {X 0,Y 374.523,Z 663.19,A -85,B 0,C 180,E1 11854.581,E2 11854.581} C_VEL
LIN {X 0,Y 372.683,Z 688.507,A -85,B 0,C 180,E1 11857.226,E2 11857.226} C_VEL
LIN {X 0,Y 370.591,Z 709.062,A -85,B 0,C 180,E1 11860.526,E2 11860.526} C_VEL
LIN {X 0,Y 368.632,Z 723.374,A -85,B 0,C 180,E1 11864.044,E2 11864.044} C_VEL
LIN {X 0,Y 367.141,Z 733.142,A -85,B 0,C 180,E1 11868.146,E2 11868.146} C_VEL
LIN {X 0,Y 366.252,Z 736.88,A -85,B 0,C 180,E1 11871.47,E2 11871.47} C_VEL
LIN {X 0,Y 365.753,Z 735.949,A -85,B 0,C 180,E1 11876.457,E2 11876.457} C_VEL
LIN {X 0,Y 365.848,Z 729.402,A -85,B 0,C 180,E1 11880.596,E2 11880.596} C_VEL
LIN {X 0,Y 366.503,Z 717.182,A -85,B 0,C 180,E1 11884.729,E2 11884.729} C_VEL
LIN {X 0,Y 367.619,Z 699.286,A -85,B 0,C 180,E1 11888.563,E2 11888.563} C_VEL
LIN {X 0,Y 369.176,Z 676.91,A -85,B 0,C 180,E1 11891.799,E2 11891.799} C_VEL
LIN {X 0,Y 370.807,Z 649.579,A -85,B 0,C 180,E1 11894.438,E2 11894.438} C_VEL
LIN {X 0,Y 371.928,Z 620.044,A -85,B 0,C 180,E1 11896.196,E2 11896.196} C_VEL
LIN {X 0,Y 371.726,Z 586.908,A -85,B 0,C 180,E1 11897.22,E2 11897.22} C_VEL
LIN {X 0,Y 362.008,Z 549.53,A -85,B 0,C 180,E1 11898.711,E2 11898.711} C_VEL
LIN {X 0,Y 361.637,Z 549.53,A -85,B 0,C 180,E1 11904.669,E2 11904.669} C_VEL
LIN {X 0,Y 361.384,Z 549.53,A -85,B 0,C 180,E1 11910.078,E2 11910.078} C_VEL
LIN {X 0,Y 361.124,Z 549.53,A -85,B 0,C 180,E1 11917.437,E2 11917.437} C_VEL
LIN {X 0,Y 361.157,Z 549.53,A -85,B 0,C 180,E1 11924.734,E2 11924.734} C_VEL
LIN {X 0,Y 361.235,Z 549.53,A -85,B 0,C 180,E1 11927.524,E2 11927.524} C_VEL
LIN {X 0,Y 363.617,Z 555.226,A -85,B 0,C 180,E1 11928.239,E2 11928.239} C_VEL
LIN {X 0,Y 381.574,Z 589.771,A -85,B 0,C 180,E1 11932.47,E2 11932.47} C_VEL
LIN {X 0,Y 392.148,Z 618.274,A -85,B 0,C 180,E1 11935.384,E2 11935.384} C_VEL
LIN {X 0,Y 392.693,Z 626.069,A -85,B 0,C 180,E1 11935.991,E2 11935.991} C_VEL
LIN {X 0,Y 387.355,Z 661.21,A -85,B 0,C 180,E1 11938.56,E2 11938.56} C_VEL
LIN {X 0,Y 381.213,Z 693.416,A -85,B 0,C 180,E1 11941.959,E2 11941.959} C_VEL
LIN {X 0,Y 375.478,Z 720.82,A -85,B 0,C 180,E1 11945.986,E2 11945.986} C_VEL
LIN {X 0,Y 370.382,Z 744.167,A -85,B 0,C 180,E1 11950.703,E2 11950.703} C_VEL
LIN {X 0,Y 366.818,Z 762.029,A -85,B 0,C 180,E1 11955.709,E2 11955.709} C_VEL
LIN {X 0,Y 364.72,Z 775.252,A -85,B 0,C 180,E1 11961.074,E2 11961.074} C_VEL
LIN {X 0,Y 363.836,Z 783.271,A -85,B 0,C 180,E1 11966.433,E2 11966.433} C_VEL
LIN {X 0,Y 363.694,Z 786.015,A -85,B 0,C 180,E1 11970,E2 11970} C_VEL
LIN {X 0,Y 363.471,Z 786.601,A -85,B 0,C 180,E1 11974.791,E2 11974.791} C_VEL
LIN {X 0,Y 363.9,Z 782.127,A -85,B 0,C 180,E1 11980.756,E2 11980.756} C_VEL
LIN {X 0,Y 365.132,Z 773.048,A -85,B 0,C 180,E1 11986.201,E2 11986.201} C_VEL
LIN {X 0,Y 367.79,Z 758.562,A -85,B 0,C 180,E1 11991.673,E2 11991.673} C_VEL
LIN {X 0,Y 372.182,Z 738.528,A -85,B 0,C 180,E1 11996.863,E2 11996.863} C_VEL
LIN {X 0,Y 378.224,Z 712.99,A -85,B 0,C 180,E1 12001.582,E2 12001.582} C_VEL
LIN {X 0,Y 384.428,Z 684.614,A -85,B 0,C 180,E1 12005.384,E2 12005.384} C_VEL
LIN {X 0,Y 390.479,Z 652.544,A -85,B 0,C 180,E1 12008.469,E2 12008.469} C_VEL
LIN {X 0,Y 394.727,Z 621.66,A -85,B 0,C 180,E1 12010.598,E2 12010.598} C_VEL
LIN {X 0,Y 386.38,Z 597.448,A -85,B 0,C 180,E1 12013.221,E2 12013.221} C_VEL
LIN {X 0,Y 369.81,Z 565.736,A -85,B 0,C 180,E1 12017.343,E2 12017.343} C_VEL
LIN {X 0,Y 361.381,Z 550.84,A -85,B 0,C 180,E1 12019.671,E2 12019.671} C_VEL
LIN {X 0,Y 361.26,Z 549.53,A -85,B 0,C 180,E1 12019.928,E2 12019.928} C_VEL
LIN {X 0,Y 361.394,Z 549.53,A -85,B 0,C 180,E1 12027.117,E2 12027.117} C_VEL
LIN {X 0,Y 361.73,Z 549.53,A -85,B 0,C 180,E1 12035.143,E2 12035.143} C_VEL
LIN {X 0,Y 370.775,Z 588.684,A -85,B 0,C 180,E1 12036.516,E2 12036.516} C_VEL
LIN {X 0,Y 370.176,Z 638.219,A -85,B 0,C 180,E1 12037.818,E2 12037.818} C_VEL
LIN {X 0,Y 369.433,Z 664.608,A -85,B 0,C 180,E1 12039.401,E2 12039.401} C_VEL
LIN {X 0,Y 368.32,Z 688.49,A -85,B 0,C 180,E1 12041.79,E2 12041.79} C_VEL
LIN {X 0,Y 367.002,Z 708.367,A -85,B 0,C 180,E1 12044.839,E2 12044.839} C_VEL
LIN {X 0,Y 366.279,Z 722.401,A -85,B 0,C 180,E1 12048.107,E2 12048.107} C_VEL
LIN {X 0,Y 365.813,Z 732.446,A -85,B 0,C 180,E1 12051.947,E2 12051.947} C_VEL
LIN {X 0,Y 365.861,Z 736.591,A -85,B 0,C 180,E1 12055.263,E2 12055.263} C_VEL
LIN {X 0,Y 365.951,Z 737.205,A -85,B 0,C 180,E1 12057.631,E2 12057.631} C_VEL
LIN {X 0,Y 366.642,Z 734.354,A -85,B 0,C 180,E1 12061.174,E2 12061.174} C_VEL
LIN {X 0,Y 367.707,Z 726.698,A -85,B 0,C 180,E1 12064.703,E2 12064.703} C_VEL
LIN {X 0,Y 369.296,Z 713.109,A -85,B 0,C 180,E1 12068.217,E2 12068.217} C_VEL
LIN {X 0,Y 371.024,Z 693.99,A -85,B 0,C 180,E1 12071.282,E2 12071.282} C_VEL
LIN {X 0,Y 372.502,Z 670.36,A -85,B 0,C 180,E1 12073.665,E2 12073.665} C_VEL
LIN {X 0,Y 373.112,Z 644.326,A -85,B 0,C 180,E1 12075.202,E2 12075.202} C_VEL
LIN {X 0,Y 373.417,Z 583.763,A -85,B 0,C 180,E1 12076.942,E2 12076.942} C_VEL
LIN {X 0,Y 364.779,Z 557.552,A -85,B 0,C 180,E1 12078.499,E2 12078.499} C_VEL
LIN {X 0,Y 361.856,Z 549.53,A -85,B 0,C 180,E1 12079.094,E2 12079.094} C_VEL
LIN {X 0,Y 361.565,Z 549.53,A -85,B 0,C 180,E1 12084.662,E2 12084.662} C_VEL
LIN {X 0,Y 361.312,Z 549.53,A -85,B 0,C 180,E1 12090.072,E2 12090.072} C_VEL
LIN {X 0,Y 361.308,Z 549.745,A -85,B 0,C 180,E1 12095.968,E2 12095.968} C_VEL
LIN {X 0,Y 363.558,Z 555.026,A -85,B 0,C 180,E1 12096.639,E2 12096.639} C_VEL
LIN {X 0,Y 379.104,Z 580.154,A -85,B 0,C 180,E1 12100.466,E2 12100.466} C_VEL
LIN {X 0,Y 394.946,Z 611.963,A -85,B 0,C 180,E1 12104.3,E2 12104.3} C_VEL
LIN {X 0,Y 401.449,Z 637.559,A -85,B 0,C 180,E1 12106.546,E2 12106.546} C_VEL
LIN {X 0,Y 394.912,Z 680.483,A -85,B 0,C 180,E1 12108.92,E2 12108.92} C_VEL
LIN {X 0,Y 387.685,Z 721.384,A -85,B 0,C 180,E1 12112.168,E2 12112.168} C_VEL
LIN {X 0,Y 381.059,Z 754.12,A -85,B 0,C 180,E1 12115.813,E2 12115.813} C_VEL
LIN {X 0,Y 374.576,Z 783.38,A -85,B 0,C 180,E1 12120.339,E2 12120.339} C_VEL
LIN {X 0,Y 369.191,Z 807.753,A -85,B 0,C 180,E1 12125.554,E2 12125.554} C_VEL
LIN {X 0,Y 365.5,Z 827.152,A -85,B 0,C 180,E1 12131.354,E2 12131.354} C_VEL
LIN {X 0,Y 363.765,Z 840.795,A -85,B 0,C 180,E1 12137.356,E2 12137.356} C_VEL
LIN {X 0,Y 363.143,Z 848.838,A -85,B 0,C 180,E1 12143.296,E2 12143.296} C_VEL
LIN {X 0,Y 360.512,Z 850.314,A -85,B 0,C 180,E1 12145.315,E2 12145.315} C_VEL
LIN {X 0,Y 355.328,Z 851.175,A -85,B 0,C 180,E1 12148.375,E2 12148.375} C_VEL
LIN {X 0,Y 355.256,Z 851.147,A -85,B 0,C 180,E1 12148.729,E2 12148.729} C_VEL
LIN {X 0,Y 355.31,Z 850.957,A -85,B 0,C 180,E1 12152.434,E2 12152.434} C_VEL
LIN {X 0,Y 355.371,Z 846.483,A -85,B 0,C 180,E1 12158.547,E2 12158.547} C_VEL
LIN {X 0,Y 356.289,Z 836.657,A -85,B 0,C 180,E1 12164.723,E2 12164.723} C_VEL
LIN {X 0,Y 358.44,Z 822.682,A -85,B 0,C 180,E1 12170.325,E2 12170.325} C_VEL
LIN {X 0,Y 362.362,Z 803.192,A -85,B 0,C 180,E1 12175.825,E2 12175.825} C_VEL
LIN {X 0,Y 368.177,Z 778.127,A -85,B 0,C 180,E1 12180.922,E2 12180.922} C_VEL
LIN {X 0,Y 374.6,Z 749.126,A -85,B 0,C 180,E1 12185.213,E2 12185.213} C_VEL
LIN {X 0,Y 381.168,Z 716.312,A -85,B 0,C 180,E1 12188.706,E2 12188.706} C_VEL
LIN {X 0,Y 388.372,Z 674.69,A -85,B 0,C 180,E1 12191.895,E2 12191.895} C_VEL
LIN {X 0,Y 393.443,Z 636.06,A -85,B 0,C 180,E1 12194.045,E2 12194.045} C_VEL
LIN {X 0,Y 385.066,Z 609.703,A -85,B 0,C 180,E1 12196.515,E2 12196.515} C_VEL
LIN {X 0,Y 368.815,Z 576.984,A -85,B 0,C 180,E1 12200.362,E2 12200.362} C_VEL
LIN {X 0,Y 353.421,Z 550.49,A -85,B 0,C 180,E1 12204.083,E2 12204.083} C_VEL
LIN {X 0,Y 353.354,Z 549.53,A -85,B 0,C 180,E1 12204.241,E2 12204.241} C_VEL
LIN {X 0,Y 353.377,Z 549.892,A -85,B 0,C 180,E1 12206.851,E2 12206.851} C_VEL
LIN {X 0,Y 364.574,Z 574.514,A -85,B 0,C 180,E1 12209.477,E2 12209.477} C_VEL
LIN {X 0,Y 369.57,Z 592.186,A -85,B 0,C 180,E1 12210.667,E2 12210.667} C_VEL
LIN {X 0,Y 368.674,Z 637.624,A -85,B 0,C 180,E1 12212.256,E2 12212.256} C_VEL
LIN {X 0,Y 367.408,Z 666.394,A -85,B 0,C 180,E1 12214.213,E2 12214.213} C_VEL
LIN {X 0,Y 365.417,Z 691.154,A -85,B 0,C 180,E1 12216.907,E2 12216.907} C_VEL
LIN {X 0,Y 363.216,Z 711.068,A -85,B 0,C 180,E1 12220.217,E2 12220.217} C_VEL
LIN {X 0,Y 360.974,Z 725.989,A -85,B 0,C 180,E1 12224.068,E2 12224.068} C_VEL
LIN {X 0,Y 359.545,Z 734.674,A -85,B 0,C 180,E1 12227.892,E2 12227.892} C_VEL
LIN {X 0,Y 358.81,Z 737.683,A -85,B 0,C 180,E1 12230.321,E2 12230.321} C_VEL
LIN {X 0,Y 358.243,Z 738.842,A -85,B 0,C 180,E1 12232.746,E2 12232.746} C_VEL
LIN {X 0,Y 357.97,Z 737.355,A -85,B 0,C 180,E1 12236.38,E2 12236.38} C_VEL
LIN {X 0,Y 358.073,Z 730.698,A -85,B 0,C 180,E1 12240.609,E2 12240.609} C_VEL
LIN {X 0,Y 358.705,Z 718.346,A -85,B 0,C 180,E1 12244.832,E2 12244.832} C_VEL
LIN {X 0,Y 359.872,Z 700.24,A -85,B 0,C 180,E1 12248.749,E2 12248.749} C_VEL
LIN {X 0,Y 361.502,Z 677.587,A -85,B 0,C 180,E1 12252.053,E2 12252.053} C_VEL
LIN {X 0,Y 363.061,Z 651.756,A -85,B 0,C 180,E1 12254.6,E2 12254.6} C_VEL
